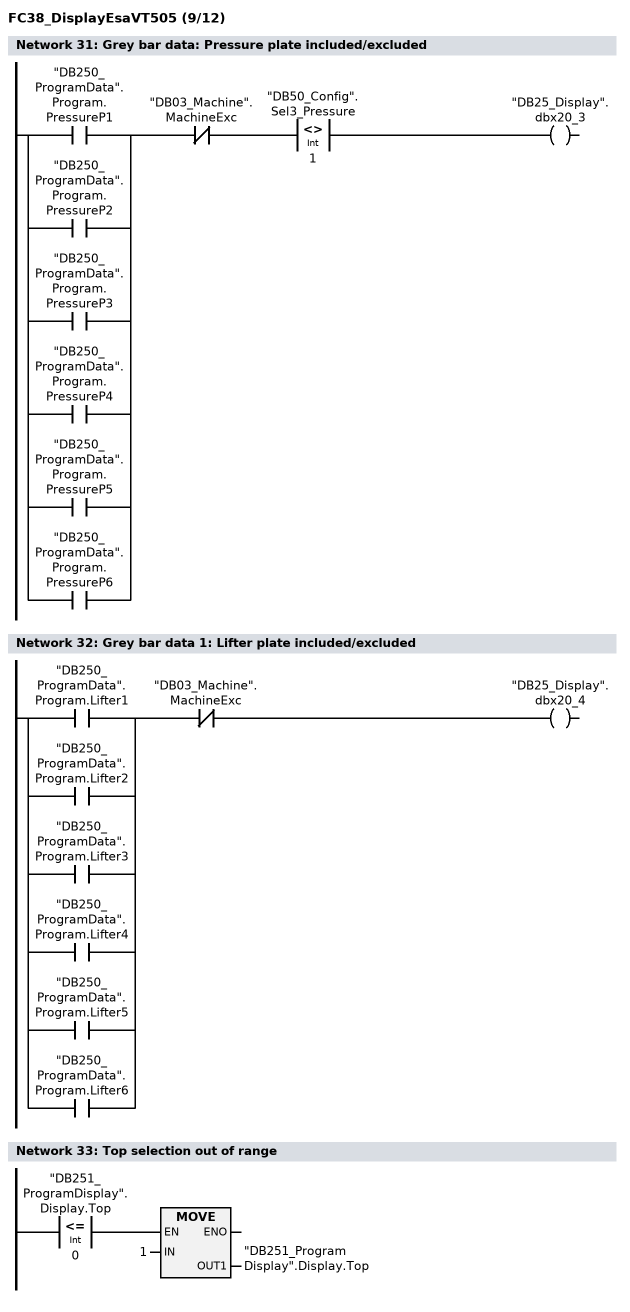
   RUNG wire#powerrail
      Contact( "DB250_ProgramData".Program.PressureP1 )
      wire#w1
      I_Contact( "DB03_Machine".MachineExc )
      { S7_Templates := "SrcType := Int" } NE_Contact(in1 := "DB50_Config".Sel3_Pressure, in2 := 1)
      Coil( "DB25_Display".dbx20_3 )
   END_RUNG
   RUNG wire#powerrail
      Contact( "DB250_ProgramData".Program.PressureP2 )
   END_RUNG wire#w1
   RUNG wire#powerrail
      Contact( "DB250_ProgramData".Program.PressureP3 )
   END_RUNG wire#w1
   RUNG wire#powerrail
      Contact( "DB250_ProgramData".Program.PressureP4 )
   END_RUNG wire#w1
   RUNG wire#powerrail
      Contact( "DB250_ProgramData".Program.PressureP5 )
   END_RUNG wire#w1
   RUNG wire#powerrail
      Contact( "DB250_ProgramData".Program.PressureP6 )
   END_RUNG wire#w1
   // the same network as SCL:
   "DB25_Display".dbx20_3 := ("DB250_ProgramData".Program.PressureP1 OR "DB250_ProgramData".Program.PressureP2 OR "DB250_ProgramData".Program.PressureP3 OR "DB250_ProgramData".Program.PressureP4 OR "DB250_ProgramData".Program.PressureP5 OR "DB250_ProgramData".Program.PressureP6) AND NOT "DB03_Machine".MachineExc AND ("DB50_Config".Sel3_Pressure <> 1);
END_REGION

REGION Network 32: Grey bar data 1: Lifter plate included/excluded
   RUNG wire#powerrail
      Contact( "DB250_ProgramData".Program.Lifter1 )
      wire#w1
      I_Contact( "DB03_Machine".MachineExc )
      Coil( "DB25_Display".dbx20_4 )
   END_RUNG
   RUNG wire#powerrail
      Contact( "DB250_ProgramData".Program.Lifter2 )
   END_RUNG wire#w1
   RUNG wire#powerrail
      Contact( "DB250_ProgramData".Program.Lifter3 )
   END_RUNG wire#w1
   RUNG wire#powerrail
      Contact( "DB250_ProgramData".Program.Lifter4 )
   END_RUNG wire#w1
   RUNG wire#powerrail
      Contact( "DB250_ProgramData".Program.Lifter5 )
   END_RUNG wire#w1
   RUNG wire#powerrail
      Contact( "DB250_ProgramData".Program.Lifter6 )
   END_RUNG wire#w1
   // the same network as SCL:
   "DB25_Display".dbx20_4 := ("DB250_ProgramData".Program.Lifter1 OR "DB250_ProgramData".Program.Lifter2 OR "DB250_ProgramData".Program.Lifter3 OR "DB250_ProgramData".Program.Lifter4 OR "DB250_ProgramData".Program.Lifter5 OR "DB250_ProgramData".Program.Lifter6) AND NOT "DB03_Machine".MachineExc;
END_REGION

REGION Network 33: Top selection out of range
   RUNG wire#powerrail
      { S7_Templates := "SrcType := Int" } LE_Contact(in1 := "DB251_ProgramDisplay".Display.Top, in2 := 0)
      { S7_GenerateENO := "TRUE" } Move(in := 1, out1 => "DB251_ProgramDisplay".Display.Top)
   END_RUNG
   // the same network as SCL:
   IF "DB251_ProgramDisplay".Display.Top <= 0 THEN "DB251_ProgramDisplay".Display.Top := 1; END_IF;
END_REGION

REGION Network 34: Top film lenght out of range
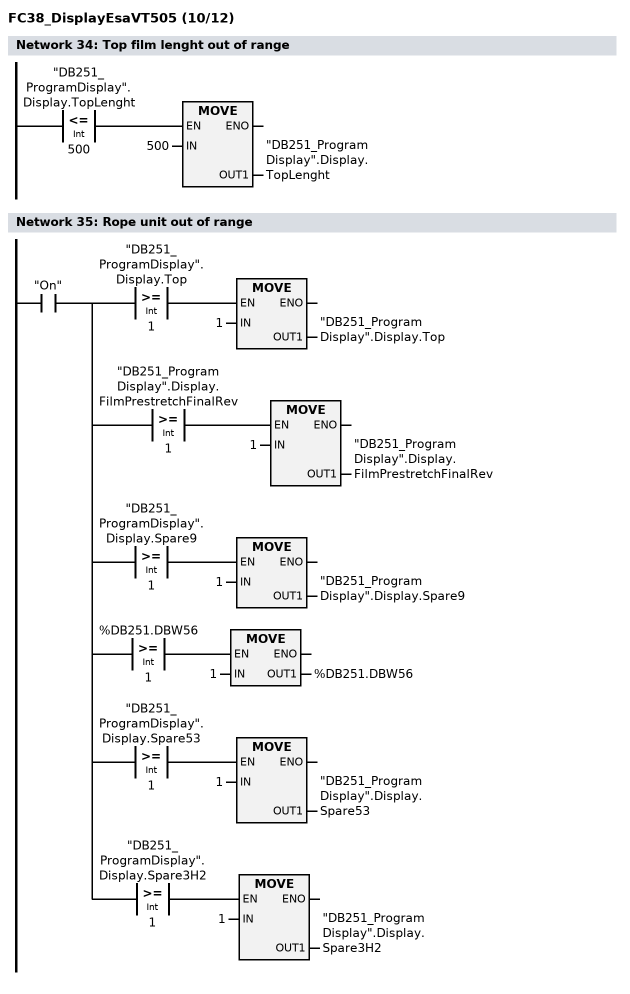
   RUNG wire#powerrail
      { S7_Templates := "SrcType := Int" } LE_Contact(in1 := "DB251_ProgramDisplay".Display.TopLenght, in2 := 500)
      { S7_GenerateENO := "TRUE" } Move(in := 500, out1 => "DB251_ProgramDisplay".Display.TopLenght)
   END_RUNG
   // the same network as SCL:
   IF "DB251_ProgramDisplay".Display.TopLenght <= 500 THEN
       "DB251_ProgramDisplay".Display.TopLenght := 500;
   END_IF;
END_REGION

REGION Network 35: Rope unit out of range
   RUNG wire#powerrail
      Contact( "On" )
      wire#w1
      { S7_Templates := "SrcType := Int" } GE_Contact(in1 := "DB251_ProgramDisplay".Display.Top, in2 := 1)
      { S7_GenerateENO := "TRUE" } Move(in := 1, out1 => "DB251_ProgramDisplay".Display.Top)
   END_RUNG
   RUNG wire#w1
      { S7_Templates := "SrcType := Int" } GE_Contact(in1 := "DB251_ProgramDisplay".Display.FilmPrestretchFinalRev, in2 := 1)
      { S7_GenerateENO := "TRUE" } Move(in := 1, out1 => "DB251_ProgramDisplay".Display.FilmPrestretchFinalRev)
   END_RUNG
   RUNG wire#w1
      { S7_Templates := "SrcType := Int" } GE_Contact(in1 := "DB251_ProgramDisplay".Display.Spare9, in2 := 1)
      { S7_GenerateENO := "TRUE" } Move(in := 1, out1 => "DB251_ProgramDisplay".Display.Spare9)
   END_RUNG
   RUNG wire#w1
      { S7_Templates := "SrcType := Int" } GE_Contact(in1 := %DB251.DBW56, in2 := 1)
      { S7_GenerateENO := "TRUE" } Move(in := 1, out1 => %DB251.DBW56)
   END_RUNG
   RUNG wire#w1
      { S7_Templates := "SrcType := Int" } GE_Contact(in1 := "DB251_ProgramDisplay".Display.Spare53, in2 := 1)
      { S7_GenerateENO := "TRUE" } Move(in := 1, out1 => "DB251_ProgramDisplay".Display.Spare53)
   END_RUNG
   RUNG wire#w1
      { S7_Templates := "SrcType := Int" } GE_Contact(in1 := "DB251_ProgramDisplay".Display.Spare3H2, in2 := 1)
      { S7_GenerateENO := "TRUE" } Move(in := 1, out1 => "DB251_ProgramDisplay".Display.Spare3H2)
   END_RUNG
   // the same network as SCL:
   IF "On" AND ("DB251_ProgramDisplay".Display.Top >= 1) THEN
       "DB251_ProgramDisplay".Display.Top := 1;
   END_IF;
   IF "On" AND ("DB251_ProgramDisplay".Display.FilmPrestretchFinalRev >= 1) THEN
       "DB251_ProgramDisplay".Display.FilmPrestretchFinalRev := 1;
   END_IF;
   IF "On" AND ("DB251_ProgramDisplay".Display.Spare9 >= 1) THEN
       "DB251_ProgramDisplay".Display.Spare9 := 1;
   END_IF;
   IF "On" AND (%DB251.DBW56 >= 1) THEN %DB251.DBW56 := 1; END_IF;
   IF "On" AND ("DB251_ProgramDisplay".Display.Spare53 >= 1) THEN
       "DB251_ProgramDisplay".Display.Spare53 := 1;
   END_IF;
   IF "On" AND ("DB251_ProgramDisplay".Display.Spare3H2 >= 1) THEN
       "DB251_ProgramDisplay".Display.Spare3H2 := 1;
   END_IF;
END_REGION

REGION Network 36: Rope unit out of range
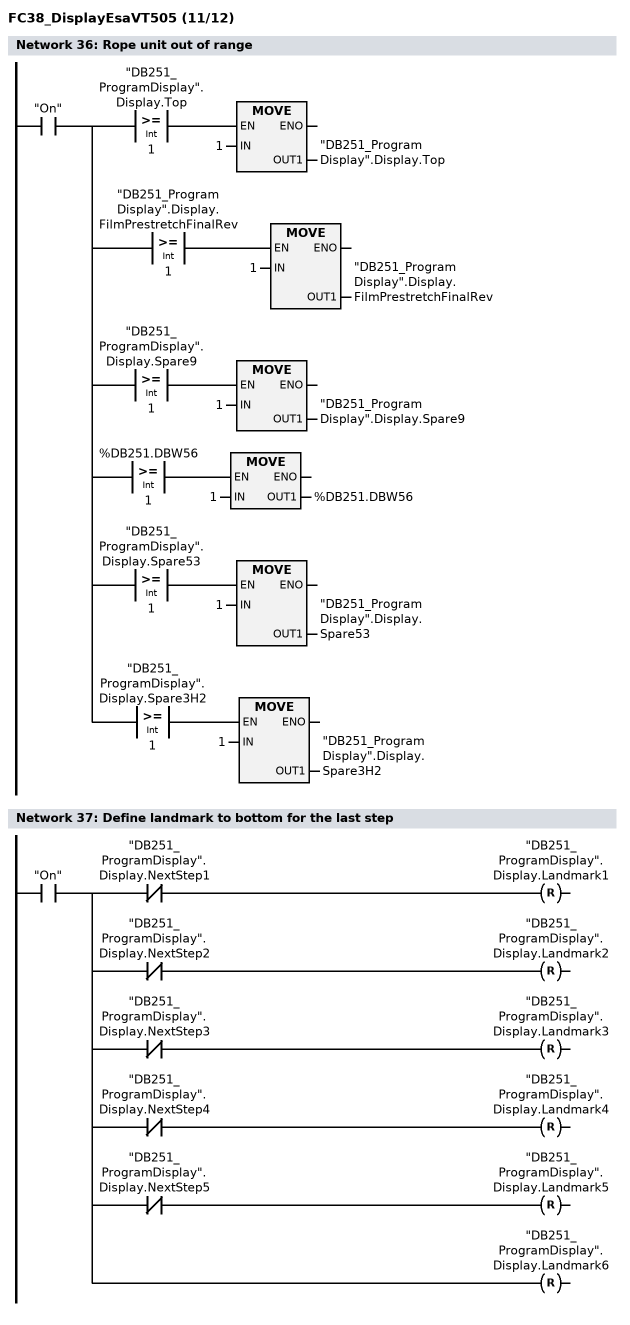
   RUNG wire#powerrail
      Contact( "On" )
      wire#w1
      { S7_Templates := "SrcType := Int" } GE_Contact(in1 := "DB251_ProgramDisplay".Display.Top, in2 := 1)
      { S7_GenerateENO := "TRUE" } Move(in := 1, out1 => "DB251_ProgramDisplay".Display.Top)
   END_RUNG
   RUNG wire#w1
      { S7_Templates := "SrcType := Int" } GE_Contact(in1 := "DB251_ProgramDisplay".Display.FilmPrestretchFinalRev, in2 := 1)
      { S7_GenerateENO := "TRUE" } Move(in := 1, out1 => "DB251_ProgramDisplay".Display.FilmPrestretchFinalRev)
   END_RUNG
   RUNG wire#w1
      { S7_Templates := "SrcType := Int" } GE_Contact(in1 := "DB251_ProgramDisplay".Display.Spare9, in2 := 1)
      { S7_GenerateENO := "TRUE" } Move(in := 1, out1 => "DB251_ProgramDisplay".Display.Spare9)
   END_RUNG
   RUNG wire#w1
      { S7_Templates := "SrcType := Int" } GE_Contact(in1 := %DB251.DBW56, in2 := 1)
      { S7_GenerateENO := "TRUE" } Move(in := 1, out1 => %DB251.DBW56)
   END_RUNG
   RUNG wire#w1
      { S7_Templates := "SrcType := Int" } GE_Contact(in1 := "DB251_ProgramDisplay".Display.Spare53, in2 := 1)
      { S7_GenerateENO := "TRUE" } Move(in := 1, out1 => "DB251_ProgramDisplay".Display.Spare53)
   END_RUNG
   RUNG wire#w1
      { S7_Templates := "SrcType := Int" } GE_Contact(in1 := "DB251_ProgramDisplay".Display.Spare3H2, in2 := 1)
      { S7_GenerateENO := "TRUE" } Move(in := 1, out1 => "DB251_ProgramDisplay".Display.Spare3H2)
   END_RUNG
   // the same network as SCL:
   IF "On" AND ("DB251_ProgramDisplay".Display.Top >= 1) THEN
       "DB251_ProgramDisplay".Display.Top := 1;
   END_IF;
   IF "On" AND ("DB251_ProgramDisplay".Display.FilmPrestretchFinalRev >= 1) THEN
       "DB251_ProgramDisplay".Display.FilmPrestretchFinalRev := 1;
   END_IF;
   IF "On" AND ("DB251_ProgramDisplay".Display.Spare9 >= 1) THEN
       "DB251_ProgramDisplay".Display.Spare9 := 1;
   END_IF;
   IF "On" AND (%DB251.DBW56 >= 1) THEN %DB251.DBW56 := 1; END_IF;
   IF "On" AND ("DB251_ProgramDisplay".Display.Spare53 >= 1) THEN
       "DB251_ProgramDisplay".Display.Spare53 := 1;
   END_IF;
   IF "On" AND ("DB251_ProgramDisplay".Display.Spare3H2 >= 1) THEN
       "DB251_ProgramDisplay".Display.Spare3H2 := 1;
   END_IF;
END_REGION

REGION Network 37: Define landmark to bottom for the last step
   RUNG wire#powerrail
      Contact( "On" )
      wire#w1
      I_Contact( "DB251_ProgramDisplay".Display.NextStep1 )
      R_Coil( "DB251_ProgramDisplay".Display.Landmark1 )
   END_RUNG
   RUNG wire#w1
      I_Contact( "DB251_ProgramDisplay".Display.NextStep2 )
      R_Coil( "DB251_ProgramDisplay".Display.Landmark2 )
   END_RUNG
   RUNG wire#w1
      I_Contact( "DB251_ProgramDisplay".Display.NextStep3 )
      R_Coil( "DB251_ProgramDisplay".Display.Landmark3 )
   END_RUNG
   RUNG wire#w1
      I_Contact( "DB251_ProgramDisplay".Display.NextStep4 )
      R_Coil( "DB251_ProgramDisplay".Display.Landmark4 )
   END_RUNG
   RUNG wire#w1
      I_Contact( "DB251_ProgramDisplay".Display.NextStep5 )
      R_Coil( "DB251_ProgramDisplay".Display.Landmark5 )
   END_RUNG
   RUNG wire#w1
      R_Coil( "DB251_ProgramDisplay".Display.Landmark6 )
   END_RUNG
   // the same network as SCL:
   IF "On" AND NOT "DB251_ProgramDisplay".Display.NextStep1 THEN
       "DB251_ProgramDisplay".Display.Landmark1 := FALSE;
   END_IF;
   IF "On" AND NOT "DB251_ProgramDisplay".Display.NextStep2 THEN
       "DB251_ProgramDisplay".Display.Landmark2 := FALSE;
   END_IF;
   IF "On" AND NOT "DB251_ProgramDisplay".Display.NextStep3 THEN
       "DB251_ProgramDisplay".Display.Landmark3 := FALSE;
   END_IF;
   IF "On" AND NOT "DB251_ProgramDisplay".Display.NextStep4 THEN
       "DB251_ProgramDisplay".Display.Landmark4 := FALSE;
   END_IF;
   IF "On" AND NOT "DB251_ProgramDisplay".Display.NextStep5 THEN
       "DB251_ProgramDisplay".Display.Landmark5 := FALSE;
   END_IF;
   IF "On" THEN "DB251_ProgramDisplay".Display.Landmark6 := FALSE; END_IF;
END_REGION

REGION Network 38
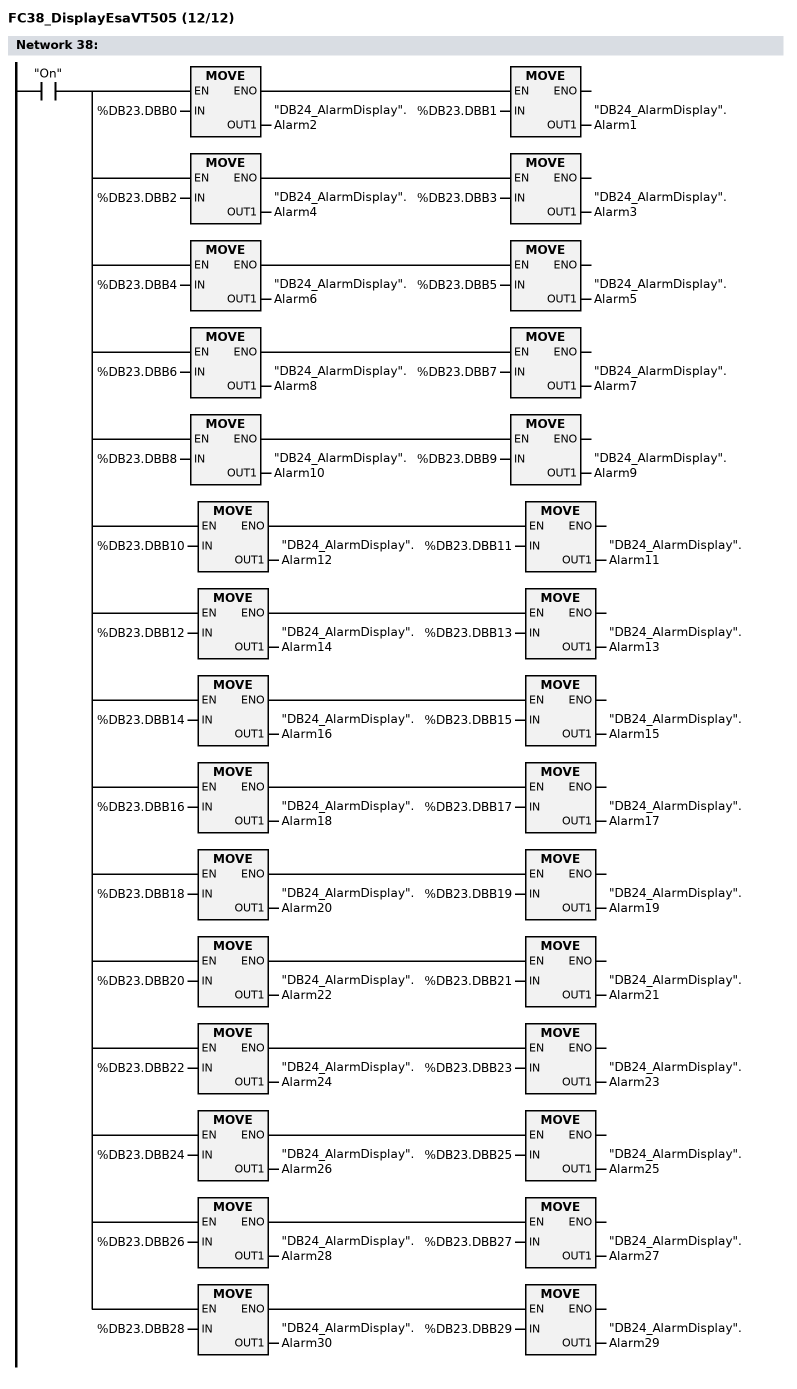
   RUNG wire#powerrail
      Contact( "On" )
      wire#w1
      { S7_GenerateENO := "TRUE" } Move(in := %DB23.DBB0, out1 => "DB24_AlarmDisplay".Alarm2)
      { S7_GenerateENO := "TRUE" } Move(in := %DB23.DBB1, out1 => "DB24_AlarmDisplay".Alarm1)
   END_RUNG
   RUNG wire#w1
      { S7_GenerateENO := "TRUE" } Move(in := %DB23.DBB2, out1 => "DB24_AlarmDisplay".Alarm4)
      { S7_GenerateENO := "TRUE" } Move(in := %DB23.DBB3, out1 => "DB24_AlarmDisplay".Alarm3)
   END_RUNG
   RUNG wire#w1
      { S7_GenerateENO := "TRUE" } Move(in := %DB23.DBB4, out1 => "DB24_AlarmDisplay".Alarm6)
      { S7_GenerateENO := "TRUE" } Move(in := %DB23.DBB5, out1 => "DB24_AlarmDisplay".Alarm5)
   END_RUNG
   RUNG wire#w1
      { S7_GenerateENO := "TRUE" } Move(in := %DB23.DBB6, out1 => "DB24_AlarmDisplay".Alarm8)
      { S7_GenerateENO := "TRUE" } Move(in := %DB23.DBB7, out1 => "DB24_AlarmDisplay".Alarm7)
   END_RUNG
   RUNG wire#w1
      { S7_GenerateENO := "TRUE" } Move(in := %DB23.DBB8, out1 => "DB24_AlarmDisplay".Alarm10)
      { S7_GenerateENO := "TRUE" } Move(in := %DB23.DBB9, out1 => "DB24_AlarmDisplay".Alarm9)
   END_RUNG
   RUNG wire#w1
      { S7_GenerateENO := "TRUE" } Move(in := %DB23.DBB10, out1 => "DB24_AlarmDisplay".Alarm12)
      { S7_GenerateENO := "TRUE" } Move(in := %DB23.DBB11, out1 => "DB24_AlarmDisplay".Alarm11)
   END_RUNG
   RUNG wire#w1
      { S7_GenerateENO := "TRUE" } Move(in := %DB23.DBB12, out1 => "DB24_AlarmDisplay".Alarm14)
      { S7_GenerateENO := "TRUE" } Move(in := %DB23.DBB13, out1 => "DB24_AlarmDisplay".Alarm13)
   END_RUNG
   RUNG wire#w1
      { S7_GenerateENO := "TRUE" } Move(in := %DB23.DBB14, out1 => "DB24_AlarmDisplay".Alarm16)
      { S7_GenerateENO := "TRUE" } Move(in := %DB23.DBB15, out1 => "DB24_AlarmDisplay".Alarm15)
   END_RUNG
   RUNG wire#w1
      { S7_GenerateENO := "TRUE" } Move(in := %DB23.DBB16, out1 => "DB24_AlarmDisplay".Alarm18)
      { S7_GenerateENO := "TRUE" } Move(in := %DB23.DBB17, out1 => "DB24_AlarmDisplay".Alarm17)
   END_RUNG
   RUNG wire#w1
      { S7_GenerateENO := "TRUE" } Move(in := %DB23.DBB18, out1 => "DB24_AlarmDisplay".Alarm20)
      { S7_GenerateENO := "TRUE" } Move(in := %DB23.DBB19, out1 => "DB24_AlarmDisplay".Alarm19)
   END_RUNG
   RUNG wire#w1
      { S7_GenerateENO := "TRUE" } Move(in := %DB23.DBB20, out1 => "DB24_AlarmDisplay".Alarm22)
      { S7_GenerateENO := "TRUE" } Move(in := %DB23.DBB21, out1 => "DB24_AlarmDisplay".Alarm21)
   END_RUNG
   RUNG wire#w1
      { S7_GenerateENO := "TRUE" } Move(in := %DB23.DBB22, out1 => "DB24_AlarmDisplay".Alarm24)
      { S7_GenerateENO := "TRUE" } Move(in := %DB23.DBB23, out1 => "DB24_AlarmDisplay".Alarm23)
   END_RUNG
   RUNG wire#w1
      { S7_GenerateENO := "TRUE" } Move(in := %DB23.DBB24, out1 => "DB24_AlarmDisplay".Alarm26)
      { S7_GenerateENO := "TRUE" } Move(in := %DB23.DBB25, out1 => "DB24_AlarmDisplay".Alarm25)
   END_RUNG
   RUNG wire#w1
      { S7_GenerateENO := "TRUE" } Move(in := %DB23.DBB26, out1 => "DB24_AlarmDisplay".Alarm28)
      { S7_GenerateENO := "TRUE" } Move(in := %DB23.DBB27, out1 => "DB24_AlarmDisplay".Alarm27)
   END_RUNG
   RUNG wire#w1
      { S7_GenerateENO := "TRUE" } Move(in := %DB23.DBB28, out1 => "DB24_AlarmDisplay".Alarm30)
      { S7_GenerateENO := "TRUE" } Move(in := %DB23.DBB29, out1 => "DB24_AlarmDisplay".Alarm29)
   END_RUNG
   // the same network as SCL:
   // ENO of a box is taken as its EN; it also drops when the box reports an error
   IF "On" THEN
       "DB24_AlarmDisplay".Alarm2 := %DB23.DBB0;
       "DB24_AlarmDisplay".Alarm1 := %DB23.DBB1;
       "DB24_AlarmDisplay".Alarm4 := %DB23.DBB2;
       "DB24_AlarmDisplay".Alarm3 := %DB23.DBB3;
       "DB24_AlarmDisplay".Alarm6 := %DB23.DBB4;
       "DB24_AlarmDisplay".Alarm5 := %DB23.DBB5;
       "DB24_AlarmDisplay".Alarm8 := %DB23.DBB6;
       "DB24_AlarmDisplay".Alarm7 := %DB23.DBB7;
       "DB24_AlarmDisplay".Alarm10 := %DB23.DBB8;
       "DB24_AlarmDisplay".Alarm9 := %DB23.DBB9;
       "DB24_AlarmDisplay".Alarm12 := %DB23.DBB10;
       "DB24_AlarmDisplay".Alarm11 := %DB23.DBB11;
       "DB24_AlarmDisplay".Alarm14 := %DB23.DBB12;
       "DB24_AlarmDisplay".Alarm13 := %DB23.DBB13;
       "DB24_AlarmDisplay".Alarm16 := %DB23.DBB14;
       "DB24_AlarmDisplay".Alarm15 := %DB23.DBB15;
       "DB24_AlarmDisplay".Alarm18 := %DB23.DBB16;
       "DB24_AlarmDisplay".Alarm17 := %DB23.DBB17;
       "DB24_AlarmDisplay".Alarm20 := %DB23.DBB18;
       "DB24_AlarmDisplay".Alarm19 := %DB23.DBB19;
       "DB24_AlarmDisplay".Alarm22 := %DB23.DBB20;
       "DB24_AlarmDisplay".Alarm21 := %DB23.DBB21;
       "DB24_AlarmDisplay".Alarm24 := %DB23.DBB22;
       "DB24_AlarmDisplay".Alarm23 := %DB23.DBB23;
       "DB24_AlarmDisplay".Alarm26 := %DB23.DBB24;
       "DB24_AlarmDisplay".Alarm25 := %DB23.DBB25;
       "DB24_AlarmDisplay".Alarm28 := %DB23.DBB26;
       "DB24_AlarmDisplay".Alarm27 := %DB23.DBB27;
       "DB24_AlarmDisplay".Alarm30 := %DB23.DBB28;
       "DB24_AlarmDisplay".Alarm29 := %DB23.DBB29;
   END_IF;
END_REGION
END_FUNCTION

FUNCTION "FC42_RopeUnit" : Void   // FC42, LAD
TITLE = RopeUnit
{ S7_Optimized_Access := 'FALSE' }
VERSION : 0.1
// stored: AutoNumber false, IsIECCheckEnabled false, SetENOAutomatically false, UDAEnableTagReadback false
   VAR_TEMP
      OpenCloseDoubleRope : Bool;
      DoubleRopeOpen : Bool;
      TempInt : Int;
      TempInt1 : Int;
   END_VAR
   VAR_TEMP   // added for the SCL form of the ladder/FBD networks
      _w1 : Bool;
   END_VAR
BEGIN

REGION Network 1: Timeout for single or lower(double) rope unit open/close
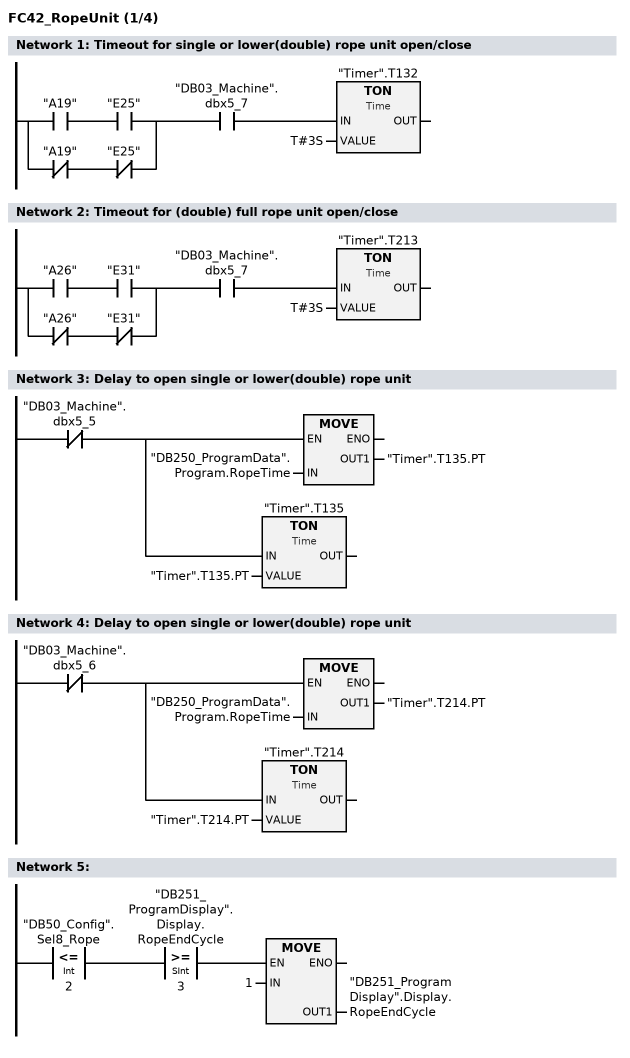
   "Timer".T132.TON(IN := (("A19" AND "E25") OR (NOT "A19" AND NOT "E25")) AND "DB03_Machine".dbx5_7, PT := T#3S);   // TON coil
END_REGION

REGION Network 2: Timeout for (double) full rope unit open/close
   "Timer".T213.TON(IN := (("A26" AND "E31") OR (NOT "A26" AND NOT "E31")) AND "DB03_Machine".dbx5_7, PT := T#3S);   // TON coil
END_REGION

REGION Network 3: Delay to open single or lower(double) rope unit
   #_w1 := NOT "DB03_Machine".dbx5_5;
   IF #_w1 THEN "Timer".T135.PT := "DB250_ProgramData".Program.RopeTime; END_IF;
   "Timer".T135.TON(IN := #_w1, PT := "Timer".T135.PT);   // TON coil
END_REGION

REGION Network 4: Delay to open single or lower(double) rope unit
   #_w1 := NOT "DB03_Machine".dbx5_6;
   IF #_w1 THEN "Timer".T214.PT := "DB250_ProgramData".Program.RopeTime; END_IF;
   "Timer".T214.TON(IN := #_w1, PT := "Timer".T214.PT);   // TON coil
END_REGION

REGION Network 5
   RUNG wire#powerrail
      { S7_Templates := "SrcType := Int" } LE_Contact(in1 := "DB50_Config".Sel8_Rope, in2 := 2)
      { S7_Templates := "SrcType := SInt" } GE_Contact(in1 := "DB251_ProgramDisplay".Display.RopeEndCycle, in2 := 3)
      { S7_GenerateENO := "TRUE" } Move(in := 1, out1 => "DB251_ProgramDisplay".Display.RopeEndCycle)
   END_RUNG
   // the same network as SCL:
   IF ("DB50_Config".Sel8_Rope <= 2) AND ("DB251_ProgramDisplay".Display.RopeEndCycle >= 3) THEN
       "DB251_ProgramDisplay".Display.RopeEndCycle := 1;
   END_IF;
END_REGION

REGION Network 6: RopeUnitOk1: Rope unit open
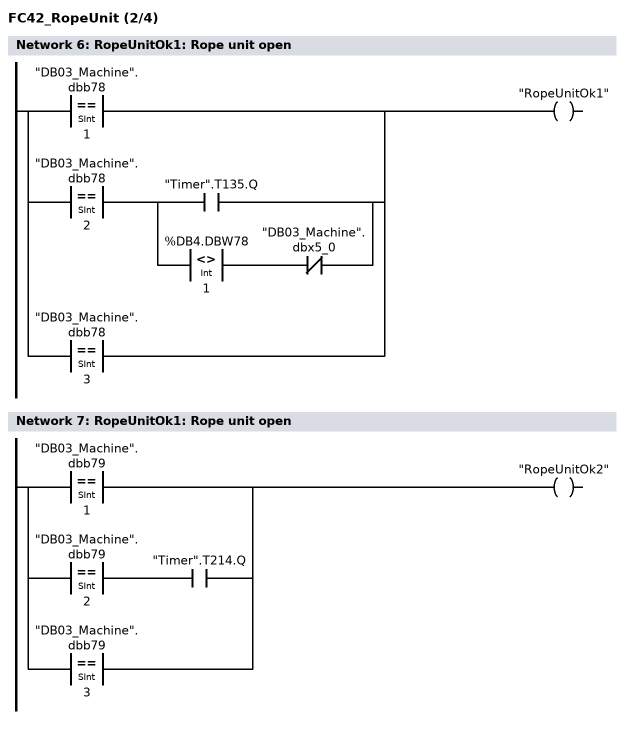
   RUNG wire#powerrail
      { S7_Templates := "SrcType := SInt" } EQ_Contact(in1 := "DB03_Machine".dbb78, in2 := 1)
      wire#w1
      Coil( "RopeUnitOk1" )
   END_RUNG
   RUNG wire#powerrail
      { S7_Templates := "SrcType := SInt" } EQ_Contact(in1 := "DB03_Machine".dbb78, in2 := 2)
      wire#w2
      Contact( "Timer".T135.Q )
   END_RUNG wire#w1
   RUNG wire#w2
      { S7_Templates := "SrcType := Int" } NE_Contact(in1 := %DB4.DBW78, in2 := 1)
      I_Contact( "DB03_Machine".dbx5_0 )
   END_RUNG wire#w1
   RUNG wire#powerrail
      { S7_Templates := "SrcType := SInt" } EQ_Contact(in1 := "DB03_Machine".dbb78, in2 := 3)
   END_RUNG wire#w1
   // the same network as SCL:
   "RopeUnitOk1" := ("DB03_Machine".dbb78 = 1) OR (("DB03_Machine".dbb78 = 2) AND ("Timer".T135.Q OR ((%DB4.DBW78 <> 1) AND NOT "DB03_Machine".dbx5_0))) OR ("DB03_Machine".dbb78 = 3);
END_REGION

REGION Network 7: RopeUnitOk1: Rope unit open
   RUNG wire#powerrail
      { S7_Templates := "SrcType := SInt" } EQ_Contact(in1 := "DB03_Machine".dbb79, in2 := 1)
      wire#w1
      Coil( "RopeUnitOk2" )
   END_RUNG
   RUNG wire#powerrail
      { S7_Templates := "SrcType := SInt" } EQ_Contact(in1 := "DB03_Machine".dbb79, in2 := 2)
      Contact( "Timer".T214.Q )
   END_RUNG wire#w1
   RUNG wire#powerrail
      { S7_Templates := "SrcType := SInt" } EQ_Contact(in1 := "DB03_Machine".dbb79, in2 := 3)
   END_RUNG wire#w1
   // the same network as SCL:
   "RopeUnitOk2" := ("DB03_Machine".dbb79 = 1) OR (("DB03_Machine".dbb79 = 2) AND "Timer".T214.Q) OR ("DB03_Machine".dbb79 = 3);
END_REGION

REGION Network 8: Closing upper(double) rope unit
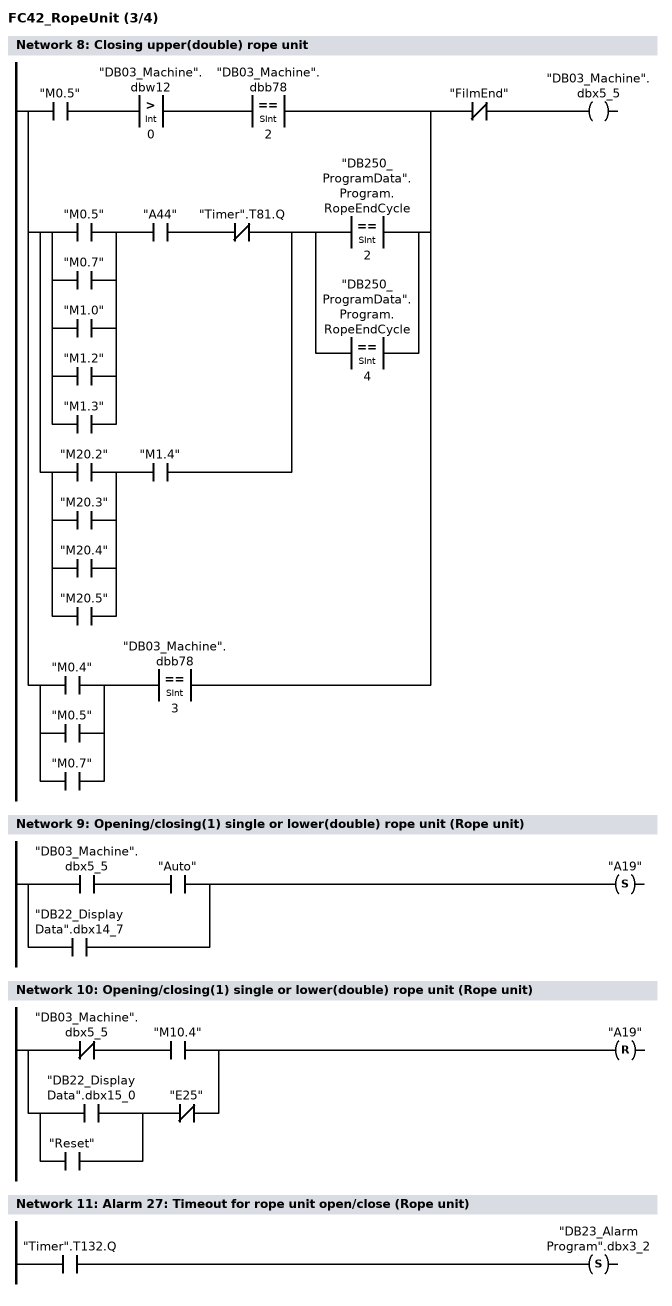
   RUNG wire#powerrail
      Contact( "M0.5" )
      { S7_Templates := "SrcType := Int" } GT_Contact(in1 := "DB03_Machine".dbw12, in2 := 0)
      { S7_Templates := "SrcType := SInt" } EQ_Contact(in1 := "DB03_Machine".dbb78, in2 := 2)
      wire#w1
      I_Contact( "FilmEnd" )
      Coil( "DB03_Machine".dbx5_5 )
   END_RUNG
   RUNG wire#powerrail
      Contact( "M0.5" )
      wire#w2
      Contact( "A44" )
      I_Contact( "Timer".T81.Q )
      wire#w3
      { S7_Templates := "SrcType := SInt" } EQ_Contact(in1 := "DB250_ProgramData".Program.RopeEndCycle, in2 := 2)
   END_RUNG wire#w1
   RUNG wire#powerrail
      Contact( "M0.7" )
   END_RUNG wire#w2
   RUNG wire#powerrail
      Contact( "M1.0" )
   END_RUNG wire#w2
   RUNG wire#powerrail
      Contact( "M1.2" )
   END_RUNG wire#w2
   RUNG wire#powerrail
      Contact( "M1.3" )
   END_RUNG wire#w2
   RUNG wire#powerrail
      Contact( "M20.2" )
      wire#w4
      Contact( "M1.4" )
   END_RUNG wire#w3
   RUNG wire#powerrail
      Contact( "M20.3" )
   END_RUNG wire#w4
   RUNG wire#powerrail
      Contact( "M20.4" )
   END_RUNG wire#w4
   RUNG wire#powerrail
      Contact( "M20.5" )
   END_RUNG wire#w4
   RUNG wire#w3
      { S7_Templates := "SrcType := SInt" } EQ_Contact(in1 := "DB250_ProgramData".Program.RopeEndCycle, in2 := 4)
   END_RUNG wire#w1
   RUNG wire#powerrail
      Contact( "M0.4" )
      wire#w5
      { S7_Templates := "SrcType := SInt" } EQ_Contact(in1 := "DB03_Machine".dbb78, in2 := 3)
   END_RUNG wire#w1
   RUNG wire#powerrail
      Contact( "M0.5" )
   END_RUNG wire#w5
   RUNG wire#powerrail
      Contact( "M0.7" )
   END_RUNG wire#w5
   // the same network as SCL:
   "DB03_Machine".dbx5_5 := (("M0.5" AND ("DB03_Machine".dbw12 > 0) AND ("DB03_Machine".dbb78 = 2)) OR (((("M0.5" OR "M0.7" OR "M1.0" OR "M1.2" OR "M1.3") AND "A44" AND NOT "Timer".T81.Q) OR (("M20.2" OR "M20.3" OR "M20.4" OR "M20.5") AND "M1.4")) AND (("DB250_ProgramData".Program.RopeEndCycle = 2) OR ("DB250_ProgramData".Program.RopeEndCycle = 4))) OR (("M0.4" OR "M0.5" OR "M0.7") AND ("DB03_Machine".dbb78 = 3))) AND NOT "FilmEnd";
END_REGION

REGION Network 9: Opening/closing(1) single or lower(double) rope unit (Rope unit)
   RUNG wire#powerrail
      Contact( "DB03_Machine".dbx5_5 )
      Contact( "Auto" )
      wire#w1
      S_Coil( "A19" )
   END_RUNG
   RUNG wire#powerrail
      Contact( "DB22_DisplayData".dbx14_7 )
   END_RUNG wire#w1
   // the same network as SCL:
   IF ("DB03_Machine".dbx5_5 AND "Auto") OR "DB22_DisplayData".dbx14_7 THEN "A19" := TRUE; END_IF;
END_REGION

REGION Network 10: Opening/closing(1) single or lower(double) rope unit (Rope unit)
   RUNG wire#powerrail
      I_Contact( "DB03_Machine".dbx5_5 )
      Contact( "M10.4" )
      wire#w1
      R_Coil( "A19" )
   END_RUNG
   RUNG wire#powerrail
      Contact( "DB22_DisplayData".dbx15_0 )
      wire#w2
      I_Contact( "E25" )
   END_RUNG wire#w1
   RUNG wire#powerrail
      Contact( "Reset" )
   END_RUNG wire#w2
   // the same network as SCL:
   IF (NOT "DB03_Machine".dbx5_5 AND "M10.4") OR (("DB22_DisplayData".dbx15_0 OR "Reset") AND NOT "E25") THEN
       "A19" := FALSE;
   END_IF;
END_REGION

REGION Network 11: Alarm 27: Timeout for rope unit open/close (Rope unit)
   RUNG wire#powerrail
      Contact( "Timer".T132.Q )
      S_Coil( "DB23_AlarmProgram".dbx3_2 )
   END_RUNG
   // the same network as SCL:
   IF "Timer".T132.Q THEN "DB23_AlarmProgram".dbx3_2 := TRUE; END_IF;
END_REGION

REGION Network 12: Closing upper(double) rope unit
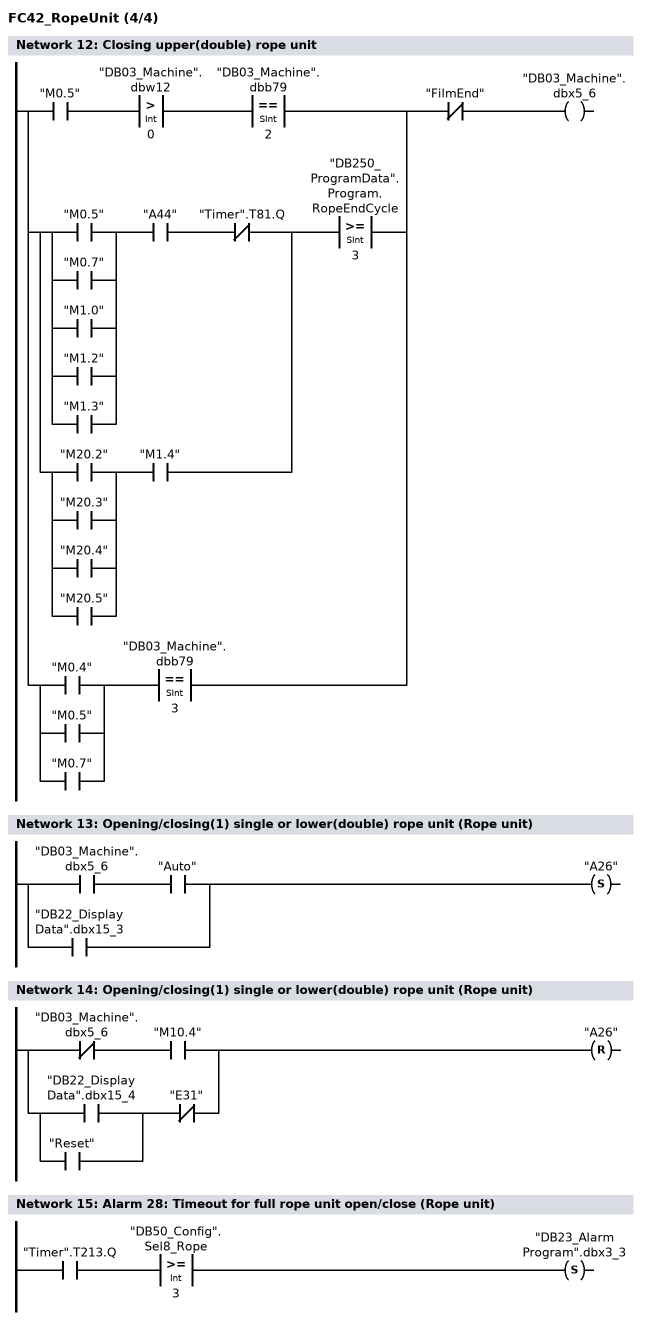
   RUNG wire#powerrail
      Contact( "M0.5" )
      { S7_Templates := "SrcType := Int" } GT_Contact(in1 := "DB03_Machine".dbw12, in2 := 0)
      { S7_Templates := "SrcType := SInt" } EQ_Contact(in1 := "DB03_Machine".dbb79, in2 := 2)
      wire#w1
      I_Contact( "FilmEnd" )
      Coil( "DB03_Machine".dbx5_6 )
   END_RUNG
   RUNG wire#powerrail
      Contact( "M0.5" )
      wire#w2
      Contact( "A44" )
      I_Contact( "Timer".T81.Q )
      wire#w3
      { S7_Templates := "SrcType := SInt" } GE_Contact(in1 := "DB250_ProgramData".Program.RopeEndCycle, in2 := 3)
   END_RUNG wire#w1
   RUNG wire#powerrail
      Contact( "M0.7" )
   END_RUNG wire#w2
   RUNG wire#powerrail
      Contact( "M1.0" )
   END_RUNG wire#w2
   RUNG wire#powerrail
      Contact( "M1.2" )
   END_RUNG wire#w2
   RUNG wire#powerrail
      Contact( "M1.3" )
   END_RUNG wire#w2
   RUNG wire#powerrail
      Contact( "M20.2" )
      wire#w4
      Contact( "M1.4" )
   END_RUNG wire#w3
   RUNG wire#powerrail
      Contact( "M20.3" )
   END_RUNG wire#w4
   RUNG wire#powerrail
      Contact( "M20.4" )
   END_RUNG wire#w4
   RUNG wire#powerrail
      Contact( "M20.5" )
   END_RUNG wire#w4
   RUNG wire#powerrail
      Contact( "M0.4" )
      wire#w5
      { S7_Templates := "SrcType := SInt" } EQ_Contact(in1 := "DB03_Machine".dbb79, in2 := 3)
   END_RUNG wire#w1
   RUNG wire#powerrail
      Contact( "M0.5" )
   END_RUNG wire#w5
   RUNG wire#powerrail
      Contact( "M0.7" )
   END_RUNG wire#w5
   // the same network as SCL:
   "DB03_Machine".dbx5_6 := (("M0.5" AND ("DB03_Machine".dbw12 > 0) AND ("DB03_Machine".dbb79 = 2)) OR (((("M0.5" OR "M0.7" OR "M1.0" OR "M1.2" OR "M1.3") AND "A44" AND NOT "Timer".T81.Q) OR (("M20.2" OR "M20.3" OR "M20.4" OR "M20.5") AND "M1.4")) AND ("DB250_ProgramData".Program.RopeEndCycle >= 3)) OR (("M0.4" OR "M0.5" OR "M0.7") AND ("DB03_Machine".dbb79 = 3))) AND NOT "FilmEnd";
END_REGION

REGION Network 13: Opening/closing(1) single or lower(double) rope unit (Rope unit)
   RUNG wire#powerrail
      Contact( "DB03_Machine".dbx5_6 )
      Contact( "Auto" )
      wire#w1
      S_Coil( "A26" )
   END_RUNG
   RUNG wire#powerrail
      Contact( "DB22_DisplayData".dbx15_3 )
   END_RUNG wire#w1
   // the same network as SCL:
   IF ("DB03_Machine".dbx5_6 AND "Auto") OR "DB22_DisplayData".dbx15_3 THEN "A26" := TRUE; END_IF;
END_REGION

REGION Network 14: Opening/closing(1) single or lower(double) rope unit (Rope unit)
   RUNG wire#powerrail
      I_Contact( "DB03_Machine".dbx5_6 )
      Contact( "M10.4" )
      wire#w1
      R_Coil( "A26" )
   END_RUNG
   RUNG wire#powerrail
      Contact( "DB22_DisplayData".dbx15_4 )
      wire#w2
      I_Contact( "E31" )
   END_RUNG wire#w1
   RUNG wire#powerrail
      Contact( "Reset" )
   END_RUNG wire#w2
   // the same network as SCL:
   IF (NOT "DB03_Machine".dbx5_6 AND "M10.4") OR (("DB22_DisplayData".dbx15_4 OR "Reset") AND NOT "E31") THEN
       "A26" := FALSE;
   END_IF;
END_REGION

REGION Network 15: Alarm 28: Timeout for full rope unit open/close (Rope unit)
   RUNG wire#powerrail
      Contact( "Timer".T213.Q )
      { S7_Templates := "SrcType := Int" } GE_Contact(in1 := "DB50_Config".Sel8_Rope, in2 := 3)
      S_Coil( "DB23_AlarmProgram".dbx3_3 )
   END_RUNG
   // the same network as SCL:
   IF "Timer".T213.Q AND ("DB50_Config".Sel8_Rope >= 3) THEN "DB23_AlarmProgram".dbx3_3 := TRUE; END_IF;
END_REGION
END_FUNCTION

FUNCTION "FC45_PrestretchPGSM_PGSA" : Void   // FC45, LAD
TITLE = Prestretch PGSM and PGSA management (HS30, Helix One)
{ S7_Optimized_Access := 'FALSE' }
AUTHOR : Robopac
VERSION : 0.0
// stored: AutoNumber false, IsIECCheckEnabled false, SetENOAutomatically false, UDAEnableTagReadback false
   VAR_TEMP
      TempInt : Int;
      TempDint : DInt;
      TempDint_2 : DInt;
      TiroStepTemp : Int;
      TiroFineTemp : Int;
   END_VAR
   VAR_TEMP   // added for the SCL form of the ladder/FBD networks
      _w1 : Bool;
      _w2 : Bool;
      _w3 : Bool;
      _w4 : Bool;
      _w5 : Bool;
      _w6 : Bool;
      _w7 : Bool;
   END_VAR
BEGIN

REGION Network 1: Film broken delay for spool carriage
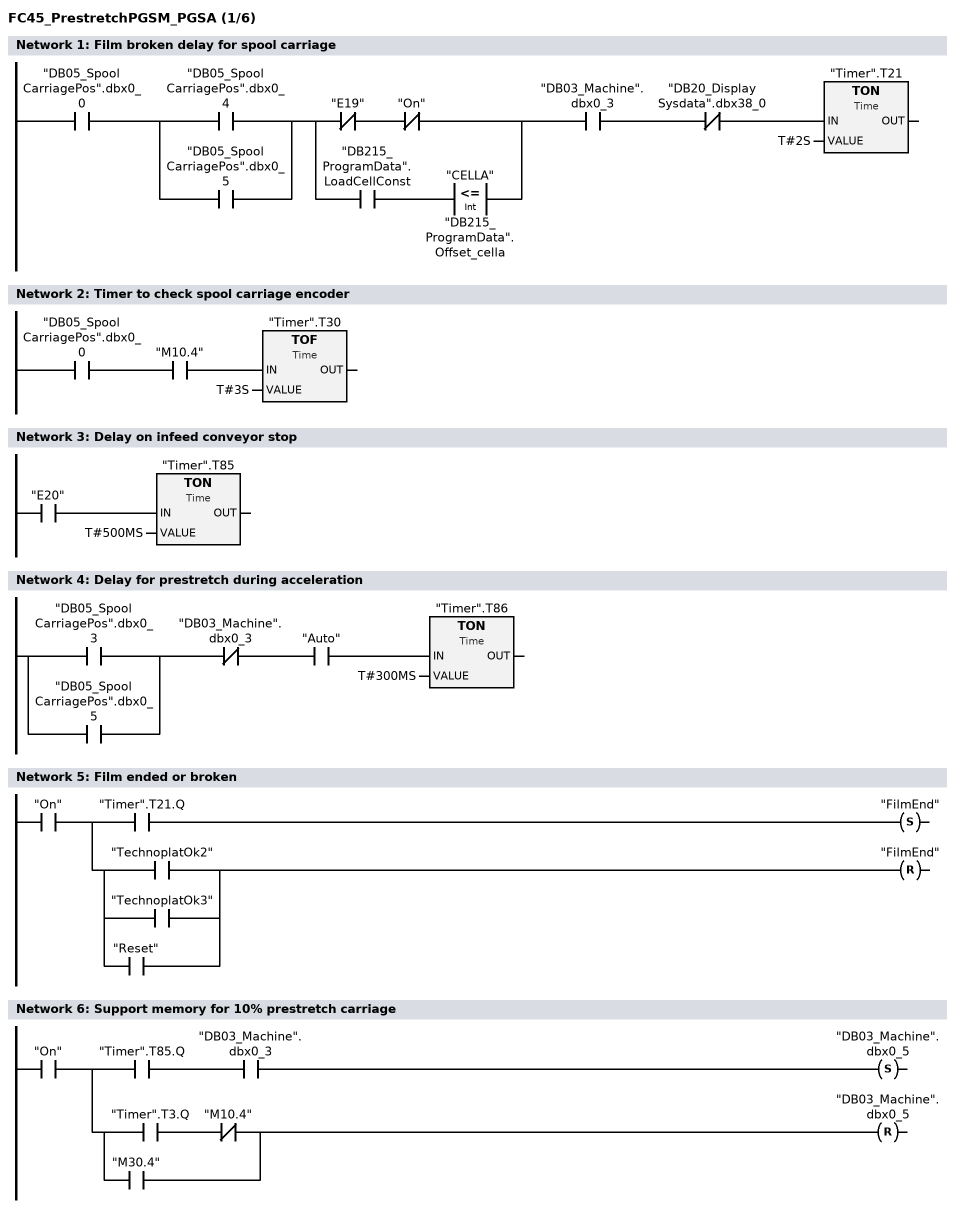
   "Timer".T21.TON(IN := "DB05_SpoolCarriagePos".dbx0_0 AND ("DB05_SpoolCarriagePos".dbx0_4 OR "DB05_SpoolCarriagePos".dbx0_5) AND ((NOT "E19" AND NOT "On") OR ("DB215_ProgramData".LoadCellConst AND ("CELLA" <= "DB215_ProgramData".Offset_cella))) AND "DB03_Machine".dbx0_3 AND NOT "DB20_DisplaySysdata".dbx38_0, PT := T#2S);   // TON coil
END_REGION

REGION Network 2: Timer to check spool carriage encoder
   "Timer".T30.TOF(IN := "DB05_SpoolCarriagePos".dbx0_0 AND "M10.4", PT := T#3S);   // TOF coil
END_REGION

REGION Network 3: Delay on infeed conveyor stop
   "Timer".T85.TON(IN := "E20", PT := T#500MS);   // TON coil
END_REGION

REGION Network 4: Delay for prestretch during acceleration
   "Timer".T86.TON(IN := ("DB05_SpoolCarriagePos".dbx0_3 OR "DB05_SpoolCarriagePos".dbx0_5) AND NOT "DB03_Machine".dbx0_3 AND "Auto", PT := T#300MS);   // TON coil
END_REGION

REGION Network 5: Film ended or broken
   RUNG wire#powerrail
      Contact( "On" )
      wire#w1
      Contact( "Timer".T21.Q )
      S_Coil( "FilmEnd" )
   END_RUNG
   RUNG wire#w1
      Contact( "TechnoplatOk2" )
      wire#w2
      R_Coil( "FilmEnd" )
   END_RUNG
   RUNG wire#w1
      Contact( "TechnoplatOk3" )
   END_RUNG wire#w2
   RUNG wire#w1
      Contact( "Reset" )
   END_RUNG wire#w2
   // the same network as SCL:
   IF "On" AND "Timer".T21.Q THEN "FilmEnd" := TRUE; END_IF;
   IF "On" AND ("TechnoplatOk2" OR "TechnoplatOk3" OR "Reset") THEN "FilmEnd" := FALSE; END_IF;
END_REGION

REGION Network 6: Support memory for 10% prestretch carriage
   RUNG wire#powerrail
      Contact( "On" )
      wire#w1
      Contact( "Timer".T85.Q )
      Contact( "DB03_Machine".dbx0_3 )
      S_Coil( "DB03_Machine".dbx0_5 )
   END_RUNG
   RUNG wire#w1
      Contact( "Timer".T3.Q )
      I_Contact( "M10.4" )
      wire#w2
      R_Coil( "DB03_Machine".dbx0_5 )
   END_RUNG
   RUNG wire#w1
      Contact( "M30.4" )
   END_RUNG wire#w2
   // the same network as SCL:
   IF "On" AND "Timer".T85.Q AND "DB03_Machine".dbx0_3 THEN "DB03_Machine".dbx0_5 := TRUE; END_IF;
   IF "On" AND (("Timer".T3.Q AND NOT "M10.4") OR "M30.4") THEN "DB03_Machine".dbx0_5 := FALSE; END_IF;
END_REGION

REGION Network 7: Support memory for prestretch PGSM or PGSA
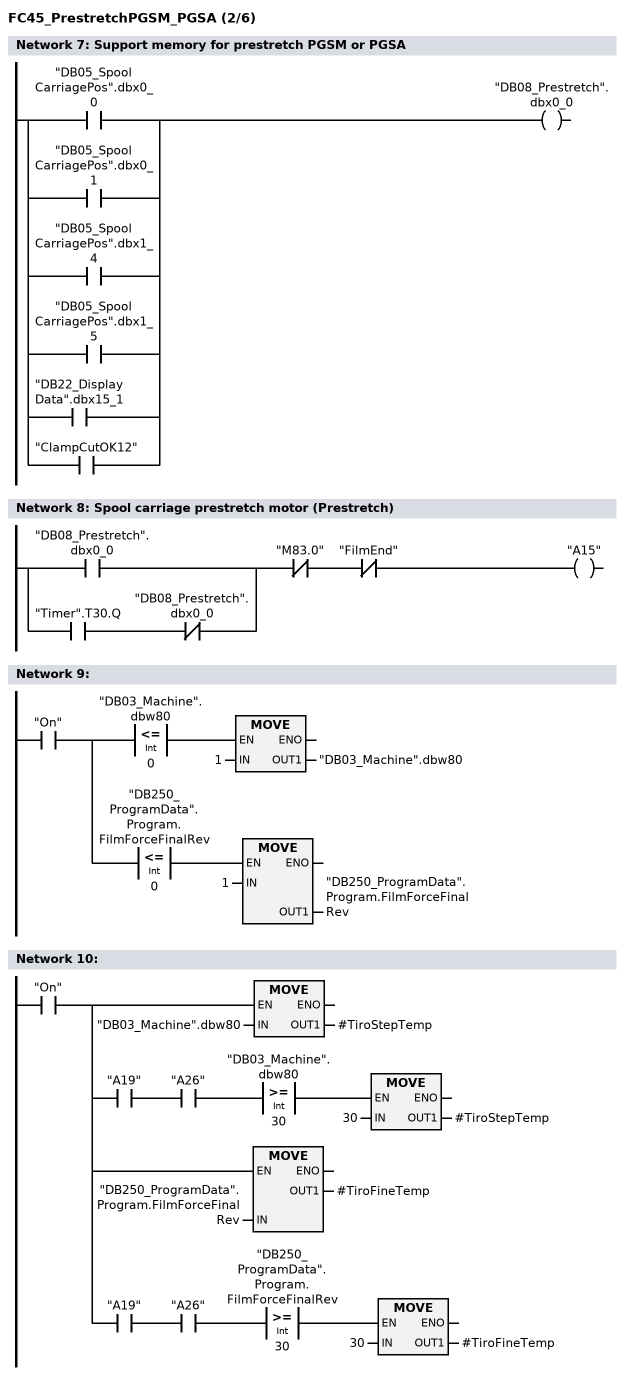
   RUNG wire#powerrail
      Contact( "DB05_SpoolCarriagePos".dbx0_0 )
      wire#w1
      Coil( "DB08_Prestretch".dbx0_0 )
   END_RUNG
   RUNG wire#powerrail
      Contact( "DB05_SpoolCarriagePos".dbx0_1 )
   END_RUNG wire#w1
   RUNG wire#powerrail
      Contact( "DB05_SpoolCarriagePos".dbx1_4 )
   END_RUNG wire#w1
   RUNG wire#powerrail
      Contact( "DB05_SpoolCarriagePos".dbx1_5 )
   END_RUNG wire#w1
   RUNG wire#powerrail
      Contact( "DB22_DisplayData".dbx15_1 )
   END_RUNG wire#w1
   RUNG wire#powerrail
      Contact( "ClampCutOK12" )
   END_RUNG wire#w1
   // the same network as SCL:
   "DB08_Prestretch".dbx0_0 := "DB05_SpoolCarriagePos".dbx0_0 OR "DB05_SpoolCarriagePos".dbx0_1 OR "DB05_SpoolCarriagePos".dbx1_4 OR "DB05_SpoolCarriagePos".dbx1_5 OR "DB22_DisplayData".dbx15_1 OR "ClampCutOK12";
END_REGION

REGION Network 8: Spool carriage prestretch motor (Prestretch)
   RUNG wire#powerrail
      Contact( "DB08_Prestretch".dbx0_0 )
      wire#w1
      I_Contact( "M83.0" )
      I_Contact( "FilmEnd" )
      Coil( "A15" )
   END_RUNG
   RUNG wire#powerrail
      Contact( "Timer".T30.Q )
      I_Contact( "DB08_Prestretch".dbx0_0 )
   END_RUNG wire#w1
   // the same network as SCL:
   "A15" := ("DB08_Prestretch".dbx0_0 OR ("Timer".T30.Q AND NOT "DB08_Prestretch".dbx0_0)) AND NOT "M83.0" AND NOT "FilmEnd";
END_REGION

REGION Network 9
   RUNG wire#powerrail
      Contact( "On" )
      wire#w1
      { S7_Templates := "SrcType := Int" } LE_Contact(in1 := "DB03_Machine".dbw80, in2 := 0)
      { S7_GenerateENO := "TRUE" } Move(in := 1, out1 => "DB03_Machine".dbw80)
   END_RUNG
   RUNG wire#w1
      { S7_Templates := "SrcType := Int" } LE_Contact(in1 := "DB250_ProgramData".Program.FilmForceFinalRev, in2 := 0)
      { S7_GenerateENO := "TRUE" } Move(in := 1, out1 => "DB250_ProgramData".Program.FilmForceFinalRev)
   END_RUNG
   // the same network as SCL:
   IF "On" AND ("DB03_Machine".dbw80 <= 0) THEN "DB03_Machine".dbw80 := 1; END_IF;
   IF "On" AND ("DB250_ProgramData".Program.FilmForceFinalRev <= 0) THEN
       "DB250_ProgramData".Program.FilmForceFinalRev := 1;
   END_IF;
END_REGION

REGION Network 10
   RUNG wire#powerrail
      Contact( "On" )
      wire#w1
      { S7_GenerateENO := "TRUE" } Move(in := "DB03_Machine".dbw80, out1 => #TiroStepTemp)
   END_RUNG
   RUNG wire#w1
      Contact( "A19" )
      Contact( "A26" )
      { S7_Templates := "SrcType := Int" } GE_Contact(in1 := "DB03_Machine".dbw80, in2 := 30)
      { S7_GenerateENO := "TRUE" } Move(in := 30, out1 => #TiroStepTemp)
   END_RUNG
   RUNG wire#w1
      { S7_GenerateENO := "TRUE" } Move(in := "DB250_ProgramData".Program.FilmForceFinalRev, out1 => #TiroFineTemp)
   END_RUNG
   RUNG wire#w1
      Contact( "A19" )
      Contact( "A26" )
      { S7_Templates := "SrcType := Int" } GE_Contact(in1 := "DB250_ProgramData".Program.FilmForceFinalRev, in2 := 30)
      { S7_GenerateENO := "TRUE" } Move(in := 30, out1 => #TiroFineTemp)
   END_RUNG
   // the same network as SCL:
   IF "On" THEN #TiroStepTemp := "DB03_Machine".dbw80; END_IF;
   IF "On" AND "A19" AND "A26" AND ("DB03_Machine".dbw80 >= 30) THEN #TiroStepTemp := 30; END_IF;
   IF "On" THEN #TiroFineTemp := "DB250_ProgramData".Program.FilmForceFinalRev; END_IF;
   IF "On" AND "A19" AND "A26" AND ("DB250_ProgramData".Program.FilmForceFinalRev >= 30) THEN
       #TiroFineTemp := 30;
   END_IF;
END_REGION

REGION Network 11
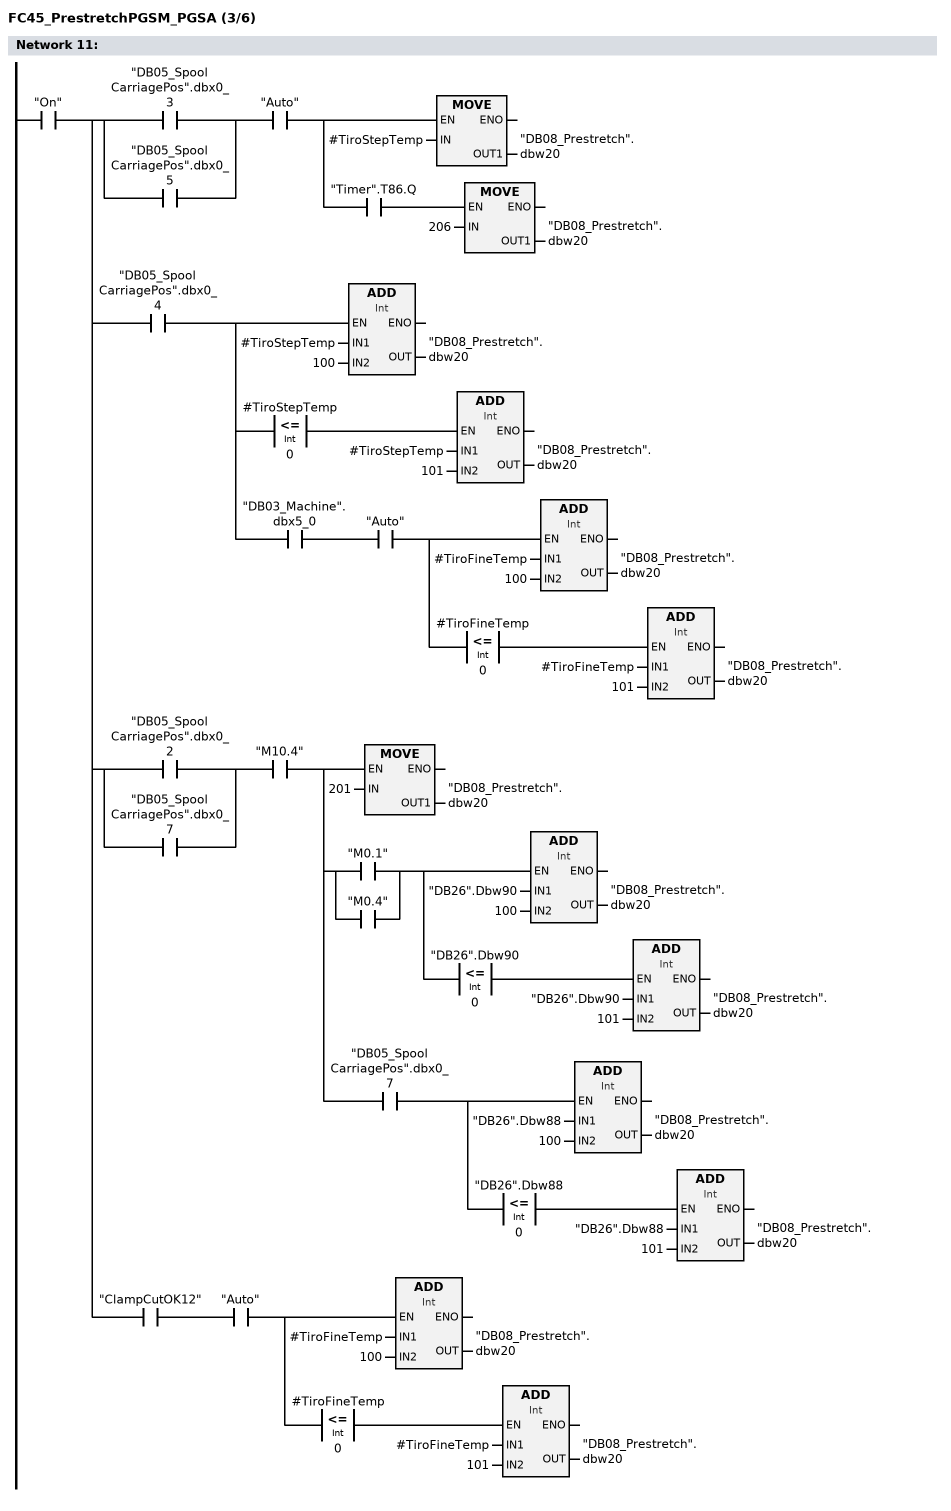
   RUNG wire#powerrail
      Contact( "On" )
      wire#w1
      Contact( "DB05_SpoolCarriagePos".dbx0_3 )
      wire#w2
      Contact( "Auto" )
      wire#w3
      { S7_GenerateENO := "TRUE" } Move(in := #TiroStepTemp, out1 => "DB08_Prestretch".dbw20)
   END_RUNG
   RUNG wire#w1
      Contact( "DB05_SpoolCarriagePos".dbx0_5 )
   END_RUNG wire#w2
   RUNG wire#w3
      Contact( "Timer".T86.Q )
      { S7_GenerateENO := "TRUE" } Move(in := 206, out1 => "DB08_Prestretch".dbw20)
   END_RUNG
   RUNG wire#w1
      Contact( "DB05_SpoolCarriagePos".dbx0_4 )
      wire#w4
      { S7_Templates := "SrcType := Int"; S7_GenerateENO := "TRUE" } Add(in1 := #TiroStepTemp, in2 := 100, out => "DB08_Prestretch".dbw20)
   END_RUNG
   RUNG wire#w4
      { S7_Templates := "SrcType := Int" } LE_Contact(in1 := #TiroStepTemp, in2 := 0)
      { S7_Templates := "SrcType := Int"; S7_GenerateENO := "TRUE" } Add(in1 := #TiroStepTemp, in2 := 101, out => "DB08_Prestretch".dbw20)
   END_RUNG
   RUNG wire#w4
      Contact( "DB03_Machine".dbx5_0 )
      Contact( "Auto" )
      wire#w5
      { S7_Templates := "SrcType := Int"; S7_GenerateENO := "TRUE" } Add(in1 := #TiroFineTemp, in2 := 100, out => "DB08_Prestretch".dbw20)
   END_RUNG
   RUNG wire#w5
      { S7_Templates := "SrcType := Int" } LE_Contact(in1 := #TiroFineTemp, in2 := 0)
      { S7_Templates := "SrcType := Int"; S7_GenerateENO := "TRUE" } Add(in1 := #TiroFineTemp, in2 := 101, out => "DB08_Prestretch".dbw20)
   END_RUNG
   RUNG wire#w1
      Contact( "DB05_SpoolCarriagePos".dbx0_2 )
      wire#w6
      Contact( "M10.4" )
      wire#w7
      { S7_GenerateENO := "TRUE" } Move(in := 201, out1 => "DB08_Prestretch".dbw20)
   END_RUNG
   RUNG wire#w1
      Contact( "DB05_SpoolCarriagePos".dbx0_7 )
   END_RUNG wire#w6
   RUNG wire#w7
      Contact( "M0.1" )
      wire#w8
      { S7_Templates := "SrcType := Int"; S7_GenerateENO := "TRUE" } Add(in1 := "DB26".Dbw90, in2 := 100, out => "DB08_Prestretch".dbw20)
   END_RUNG
   RUNG wire#w7
      Contact( "M0.4" )
   END_RUNG wire#w8
   RUNG wire#w8
      { S7_Templates := "SrcType := Int" } LE_Contact(in1 := "DB26".Dbw90, in2 := 0)
      { S7_Templates := "SrcType := Int"; S7_GenerateENO := "TRUE" } Add(in1 := "DB26".Dbw90, in2 := 101, out => "DB08_Prestretch".dbw20)
   END_RUNG
   RUNG wire#w7
      Contact( "DB05_SpoolCarriagePos".dbx0_7 )
      wire#w9
      { S7_Templates := "SrcType := Int"; S7_GenerateENO := "TRUE" } Add(in1 := "DB26".Dbw88, in2 := 100, out => "DB08_Prestretch".dbw20)
   END_RUNG
   RUNG wire#w9
      { S7_Templates := "SrcType := Int" } LE_Contact(in1 := "DB26".Dbw88, in2 := 0)
      { S7_Templates := "SrcType := Int"; S7_GenerateENO := "TRUE" } Add(in1 := "DB26".Dbw88, in2 := 101, out => "DB08_Prestretch".dbw20)
   END_RUNG
   RUNG wire#w1
      Contact( "ClampCutOK12" )
      Contact( "Auto" )
      wire#w10
      { S7_Templates := "SrcType := Int"; S7_GenerateENO := "TRUE" } Add(in1 := #TiroFineTemp, in2 := 100, out => "DB08_Prestretch".dbw20)
   END_RUNG
   RUNG wire#w10
      { S7_Templates := "SrcType := Int" } LE_Contact(in1 := #TiroFineTemp, in2 := 0)
      { S7_Templates := "SrcType := Int"; S7_GenerateENO := "TRUE" } Add(in1 := #TiroFineTemp, in2 := 101, out => "DB08_Prestretch".dbw20)
   END_RUNG
   // the same network as SCL:
   #_w1 := "On" AND ("DB05_SpoolCarriagePos".dbx0_3 OR "DB05_SpoolCarriagePos".dbx0_5) AND "Auto";
   IF #_w1 THEN "DB08_Prestretch".dbw20 := #TiroStepTemp; END_IF;
   IF #_w1 AND "Timer".T86.Q THEN "DB08_Prestretch".dbw20 := 206; END_IF;
   #_w2 := "On" AND "DB05_SpoolCarriagePos".dbx0_4;
   IF #_w2 THEN "DB08_Prestretch".dbw20 := #TiroStepTemp + 100; END_IF;
   IF #_w2 AND (#TiroStepTemp <= 0) THEN "DB08_Prestretch".dbw20 := #TiroStepTemp + 101; END_IF;
   #_w3 := #_w2 AND "DB03_Machine".dbx5_0 AND "Auto";
   IF #_w3 THEN "DB08_Prestretch".dbw20 := #TiroFineTemp + 100; END_IF;
   IF #_w3 AND (#TiroFineTemp <= 0) THEN "DB08_Prestretch".dbw20 := #TiroFineTemp + 101; END_IF;
   #_w4 := "On" AND ("DB05_SpoolCarriagePos".dbx0_2 OR "DB05_SpoolCarriagePos".dbx0_7) AND "M10.4";
   IF #_w4 THEN "DB08_Prestretch".dbw20 := 201; END_IF;
   #_w5 := #_w4 AND ("M0.1" OR "M0.4");
   IF #_w5 THEN "DB08_Prestretch".dbw20 := "DB26".Dbw90 + 100; END_IF;
   IF #_w5 AND ("DB26".Dbw90 <= 0) THEN "DB08_Prestretch".dbw20 := "DB26".Dbw90 + 101; END_IF;
   #_w6 := #_w4 AND "DB05_SpoolCarriagePos".dbx0_7;
   IF #_w6 THEN "DB08_Prestretch".dbw20 := "DB26".Dbw88 + 100; END_IF;
   IF #_w6 AND ("DB26".Dbw88 <= 0) THEN "DB08_Prestretch".dbw20 := "DB26".Dbw88 + 101; END_IF;
   #_w7 := "On" AND "ClampCutOK12" AND "Auto";
   IF #_w7 THEN "DB08_Prestretch".dbw20 := #TiroFineTemp + 100; END_IF;
   IF #_w7 AND (#TiroFineTemp <= 0) THEN "DB08_Prestretch".dbw20 := #TiroFineTemp + 101; END_IF;
END_REGION

REGION Network 12
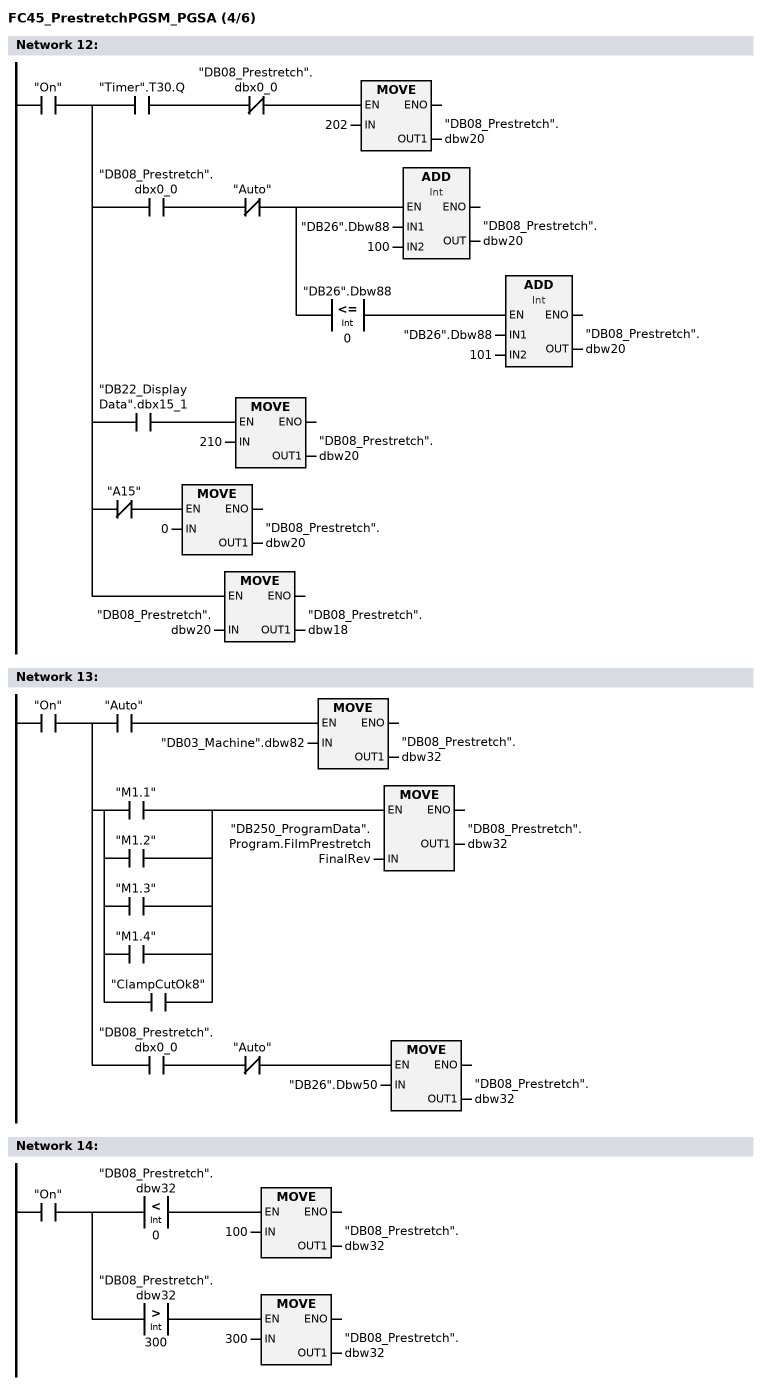
   RUNG wire#powerrail
      Contact( "On" )
      wire#w1
      Contact( "Timer".T30.Q )
      I_Contact( "DB08_Prestretch".dbx0_0 )
      { S7_GenerateENO := "TRUE" } Move(in := 202, out1 => "DB08_Prestretch".dbw20)
   END_RUNG
   RUNG wire#w1
      Contact( "DB08_Prestretch".dbx0_0 )
      I_Contact( "Auto" )
      wire#w2
      { S7_Templates := "SrcType := Int"; S7_GenerateENO := "TRUE" } Add(in1 := "DB26".Dbw88, in2 := 100, out => "DB08_Prestretch".dbw20)
   END_RUNG
   RUNG wire#w2
      { S7_Templates := "SrcType := Int" } LE_Contact(in1 := "DB26".Dbw88, in2 := 0)
      { S7_Templates := "SrcType := Int"; S7_GenerateENO := "TRUE" } Add(in1 := "DB26".Dbw88, in2 := 101, out => "DB08_Prestretch".dbw20)
   END_RUNG
   RUNG wire#w1
      Contact( "DB22_DisplayData".dbx15_1 )
      { S7_GenerateENO := "TRUE" } Move(in := 210, out1 => "DB08_Prestretch".dbw20)
   END_RUNG
   RUNG wire#w1
      I_Contact( "A15" )
      { S7_GenerateENO := "TRUE" } Move(in := 0, out1 => "DB08_Prestretch".dbw20)
   END_RUNG
   RUNG wire#w1
      { S7_GenerateENO := "TRUE" } Move(in := "DB08_Prestretch".dbw20, out1 => "DB08_Prestretch".dbw18)
   END_RUNG
   // the same network as SCL:
   IF "On" AND "Timer".T30.Q AND NOT "DB08_Prestretch".dbx0_0 THEN "DB08_Prestretch".dbw20 := 202; END_IF;
   #_w1 := "On" AND "DB08_Prestretch".dbx0_0 AND NOT "Auto";
   IF #_w1 THEN "DB08_Prestretch".dbw20 := "DB26".Dbw88 + 100; END_IF;
   IF #_w1 AND ("DB26".Dbw88 <= 0) THEN "DB08_Prestretch".dbw20 := "DB26".Dbw88 + 101; END_IF;
   IF "On" AND "DB22_DisplayData".dbx15_1 THEN "DB08_Prestretch".dbw20 := 210; END_IF;
   IF "On" AND NOT "A15" THEN "DB08_Prestretch".dbw20 := 0; END_IF;
   IF "On" THEN "DB08_Prestretch".dbw18 := "DB08_Prestretch".dbw20; END_IF;
END_REGION

REGION Network 13
   RUNG wire#powerrail
      Contact( "On" )
      wire#w1
      Contact( "Auto" )
      { S7_GenerateENO := "TRUE" } Move(in := "DB03_Machine".dbw82, out1 => "DB08_Prestretch".dbw32)
   END_RUNG
   RUNG wire#w1
      Contact( "M1.1" )
      wire#w2
      { S7_GenerateENO := "TRUE" } Move(in := "DB250_ProgramData".Program.FilmPrestretchFinalRev, out1 => "DB08_Prestretch".dbw32)
   END_RUNG
   RUNG wire#w1
      Contact( "M1.2" )
   END_RUNG wire#w2
   RUNG wire#w1
      Contact( "M1.3" )
   END_RUNG wire#w2
   RUNG wire#w1
      Contact( "M1.4" )
   END_RUNG wire#w2
   RUNG wire#w1
      Contact( "ClampCutOk8" )
   END_RUNG wire#w2
   RUNG wire#w1
      Contact( "DB08_Prestretch".dbx0_0 )
      I_Contact( "Auto" )
      { S7_GenerateENO := "TRUE" } Move(in := "DB26".Dbw50, out1 => "DB08_Prestretch".dbw32)
   END_RUNG
   // the same network as SCL:
   IF "On" AND "Auto" THEN "DB08_Prestretch".dbw32 := "DB03_Machine".dbw82; END_IF;
   IF "On" AND ("M1.1" OR "M1.2" OR "M1.3" OR "M1.4" OR "ClampCutOk8") THEN
       "DB08_Prestretch".dbw32 := "DB250_ProgramData".Program.FilmPrestretchFinalRev;
   END_IF;
   IF "On" AND "DB08_Prestretch".dbx0_0 AND NOT "Auto" THEN "DB08_Prestretch".dbw32 := "DB26".Dbw50; END_IF;
END_REGION

REGION Network 14
   RUNG wire#powerrail
      Contact( "On" )
      wire#w1
      { S7_Templates := "SrcType := Int" } LT_Contact(in1 := "DB08_Prestretch".dbw32, in2 := 0)
      { S7_GenerateENO := "TRUE" } Move(in := 100, out1 => "DB08_Prestretch".dbw32)
   END_RUNG
   RUNG wire#w1
      { S7_Templates := "SrcType := Int" } GT_Contact(in1 := "DB08_Prestretch".dbw32, in2 := 300)
      { S7_GenerateENO := "TRUE" } Move(in := 300, out1 => "DB08_Prestretch".dbw32)
   END_RUNG
   // the same network as SCL:
   IF "On" AND ("DB08_Prestretch".dbw32 < 0) THEN "DB08_Prestretch".dbw32 := 100; END_IF;
   IF "On" AND ("DB08_Prestretch".dbw32 > 300) THEN "DB08_Prestretch".dbw32 := 300; END_IF;
END_REGION

REGION Network 15
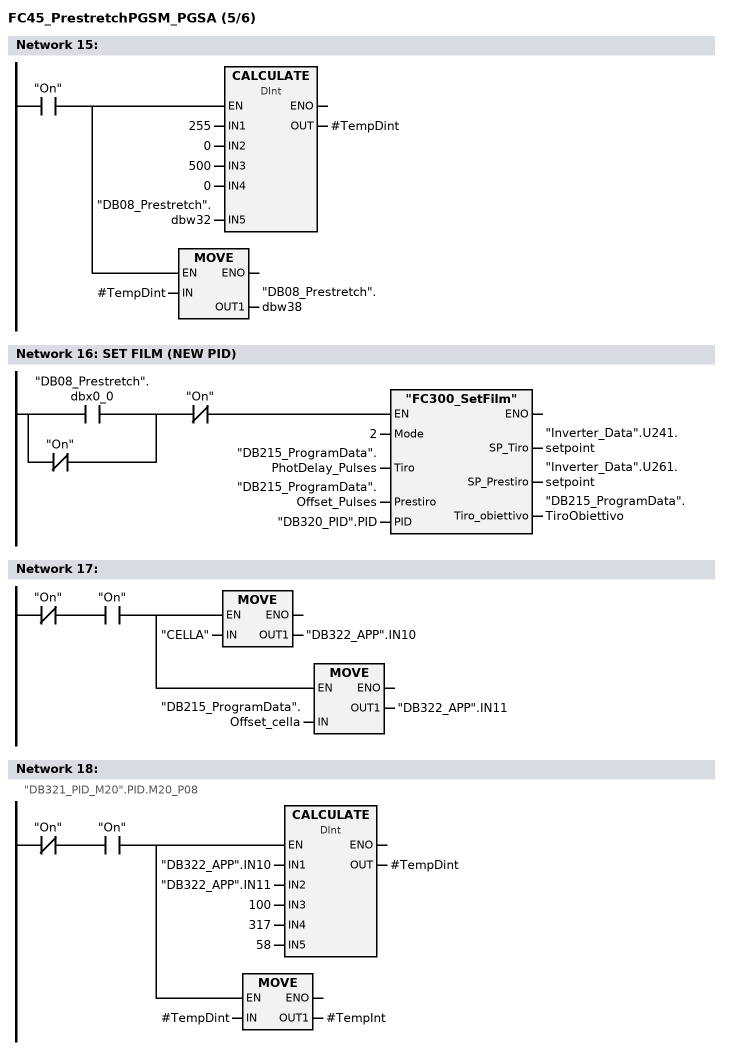
   RUNG wire#powerrail
      Contact( "On" )
      wire#w1
      { S7_Templates := "SrcType := DInt"; S7_GenerateENO := "TRUE"; S7_Expression := "((IN5-IN4)*(IN1-IN2)/(IN3-IN4))+IN2" } Calculate(in1 := 255, in2 := 0, in3 := 500, in4 := 0, in5 := "DB08_Prestretch".dbw32, out => #TempDint)
   END_RUNG
   RUNG wire#w1
      { S7_GenerateENO := "TRUE" } Move(in := #TempDint, out1 => "DB08_Prestretch".dbw38)
   END_RUNG
   // the same network as SCL:
   IF "On" THEN
       #TempDint := (("DB08_Prestretch".dbw32-0)*(255-0)/(500-0))+0;
       "DB08_Prestretch".dbw38 := #TempDint;
   END_IF;
END_REGION

REGION Network 16: SET FILM (NEW PID)
   RUNG wire#powerrail
      Contact( "DB08_Prestretch".dbx0_0 )
      wire#w1
      I_Contact( "On" )
      "FC300_SetFilm"(Mode := 2, Tiro := "DB215_ProgramData".PhotDelay_Pulses, Prestiro := "DB215_ProgramData".Offset_Pulses, PID := "DB320_PID".PID, SP_Tiro => "Inverter_Data".U241.setpoint, SP_Prestiro => "Inverter_Data".U261.setpoint, Tiro_obiettivo => "DB215_ProgramData".TiroObiettivo)
   END_RUNG
   RUNG wire#powerrail
      I_Contact( "On" )
   END_RUNG wire#w1
   // the same network as SCL:
   IF ("DB08_Prestretch".dbx0_0 OR NOT "On") AND NOT "On" THEN
       "FC300_SetFilm"(Mode := 2,
                       Tiro := "DB215_ProgramData".PhotDelay_Pulses,
                       Prestiro := "DB215_ProgramData".Offset_Pulses,
                       PID := "DB320_PID".PID,
                       SP_Tiro => "Inverter_Data".U241.setpoint,
                       SP_Prestiro => "Inverter_Data".U261.setpoint,
                       Tiro_obiettivo => "DB215_ProgramData".TiroObiettivo);
   END_IF;
END_REGION

REGION Network 17
   RUNG wire#powerrail
      I_Contact( "On" )
      Contact( "On" )
      wire#w1
      Move(in := "CELLA", out1 => "DB322_APP".IN10)
   END_RUNG
   RUNG wire#w1
      Move(in := "DB215_ProgramData".Offset_cella, out1 => "DB322_APP".IN11)
   END_RUNG
   // the same network as SCL:
   IF NOT "On" AND "On" THEN
       "DB322_APP".IN10 := "CELLA";
       "DB322_APP".IN11 := "DB215_ProgramData".Offset_cella;
   END_IF;
END_REGION

REGION Network 18
   // "DB321_PID_M20".PID.M20_P08
   RUNG wire#powerrail
      I_Contact( "On" )
      Contact( "On" )
      wire#w1
      { S7_Templates := "SrcType := DInt"; S7_Expression := "((IN1-IN2)*IN3/IN4)+IN5" } Calculate(in1 := "DB322_APP".IN10, in2 := "DB322_APP".IN11, in3 := 100, in4 := 317, in5 := 58, out => #TempDint)
   END_RUNG
   RUNG wire#w1
      Move(in := #TempDint, out1 => #TempInt)
   END_RUNG
   // the same network as SCL:
   IF NOT "On" AND "On" THEN
       #TempDint := (("DB322_APP".IN10-"DB322_APP".IN11)*100/317)+58;
       #TempInt := #TempDint;
   END_IF;
END_REGION

REGION Network 19
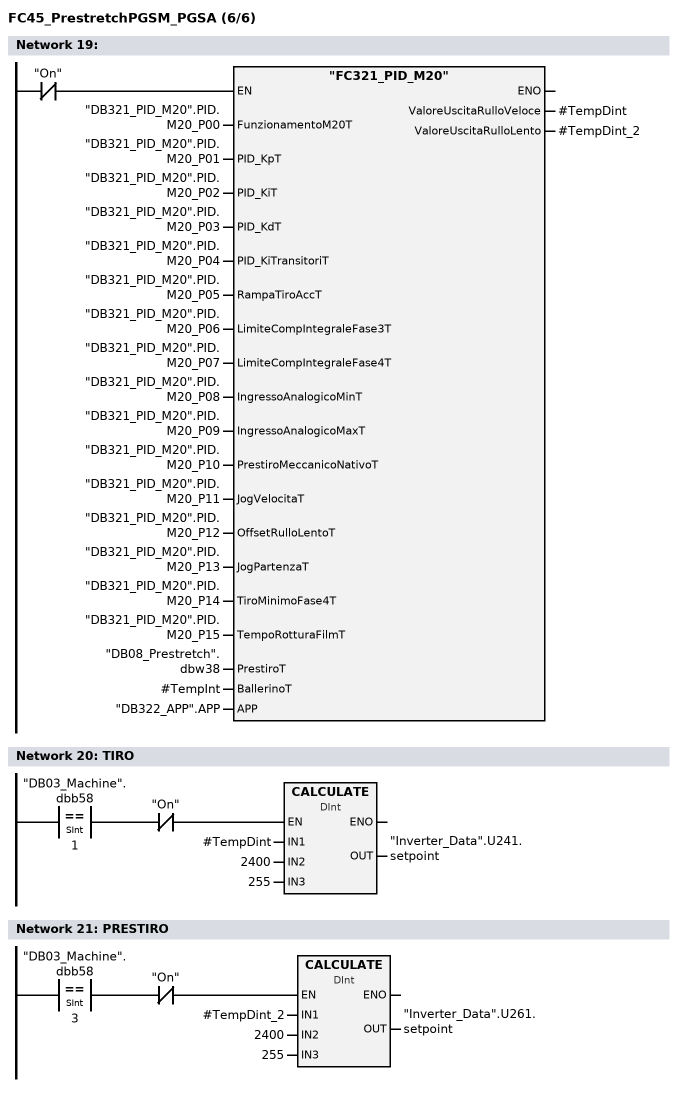
   RUNG wire#powerrail
      I_Contact( "On" )
      "FC321_PID_M20"(FunzionamentoM20T := "DB321_PID_M20".PID.M20_P00, PID_KpT := "DB321_PID_M20".PID.M20_P01, PID_KiT := "DB321_PID_M20".PID.M20_P02, PID_KdT := "DB321_PID_M20".PID.M20_P03, PID_KiTransitoriT := "DB321_PID_M20".PID.M20_P04, RampaTiroAccT := "DB321_PID_M20".PID.M20_P05, LimiteCompIntegraleFase3T := "DB321_PID_M20".PID.M20_P06, LimiteCompIntegraleFase4T := "DB321_PID_M20".PID.M20_P07, IngressoAnalogicoMinT := "DB321_PID_M20".PID.M20_P08, IngressoAnalogicoMaxT := "DB321_PID_M20".PID.M20_P09, PrestiroMeccanicoNativoT := "DB321_PID_M20".PID.M20_P10, JogVelocitaT := "DB321_PID_M20".PID.M20_P11, OffsetRulloLentoT := "DB321_PID_M20".PID.M20_P12, JogPartenzaT := "DB321_PID_M20".PID.M20_P13, TiroMinimoFase4T := "DB321_PID_M20".PID.M20_P14, TempoRotturaFilmT := "DB321_PID_M20".PID.M20_P15, PrestiroT := "DB08_Prestretch".dbw38, BallerinoT := #TempInt, APP := "DB322_APP".APP, ValoreUscitaRulloVeloce => #TempDint, ValoreUscitaRulloLento => #TempDint_2)
   END_RUNG
   // the same network as SCL:
   IF NOT "On" THEN
       "FC321_PID_M20"(FunzionamentoM20T := "DB321_PID_M20".PID.M20_P00,
                       PID_KpT := "DB321_PID_M20".PID.M20_P01,
                       PID_KiT := "DB321_PID_M20".PID.M20_P02,
                       PID_KdT := "DB321_PID_M20".PID.M20_P03,
                       PID_KiTransitoriT := "DB321_PID_M20".PID.M20_P04,
                       RampaTiroAccT := "DB321_PID_M20".PID.M20_P05,
                       LimiteCompIntegraleFase3T := "DB321_PID_M20".PID.M20_P06,
                       LimiteCompIntegraleFase4T := "DB321_PID_M20".PID.M20_P07,
                       IngressoAnalogicoMinT := "DB321_PID_M20".PID.M20_P08,
                       IngressoAnalogicoMaxT := "DB321_PID_M20".PID.M20_P09,
                       PrestiroMeccanicoNativoT := "DB321_PID_M20".PID.M20_P10,
                       JogVelocitaT := "DB321_PID_M20".PID.M20_P11,
                       OffsetRulloLentoT := "DB321_PID_M20".PID.M20_P12,
                       JogPartenzaT := "DB321_PID_M20".PID.M20_P13,
                       TiroMinimoFase4T := "DB321_PID_M20".PID.M20_P14,
                       TempoRotturaFilmT := "DB321_PID_M20".PID.M20_P15,
                       PrestiroT := "DB08_Prestretch".dbw38,
                       BallerinoT := #TempInt,
                       APP := "DB322_APP".APP,
                       ValoreUscitaRulloVeloce => #TempDint,
                       ValoreUscitaRulloLento => #TempDint_2);
   END_IF;
END_REGION

REGION Network 20: TIRO
   RUNG wire#powerrail
      { S7_Templates := "SrcType := SInt" } EQ_Contact(in1 := "DB03_Machine".dbb58, in2 := 1)
      I_Contact( "On" )
      { S7_Templates := "SrcType := DInt"; S7_Expression := "IN1*IN2/IN3" } Calculate(in1 := #TempDint, in2 := 2400, in3 := 255, out => "Inverter_Data".U241.setpoint)
   END_RUNG
   // the same network as SCL:
   IF ("DB03_Machine".dbb58 = 1) AND NOT "On" THEN
       "Inverter_Data".U241.setpoint := #TempDint*2400/255;
   END_IF;
END_REGION

REGION Network 21: PRESTIRO
   RUNG wire#powerrail
      { S7_Templates := "SrcType := SInt" } EQ_Contact(in1 := "DB03_Machine".dbb58, in2 := 3)
      I_Contact( "On" )
      { S7_Templates := "SrcType := DInt"; S7_Expression := "IN1*IN2/IN3" } Calculate(in1 := #TempDint_2, in2 := 2400, in3 := 255, out => "Inverter_Data".U261.setpoint)
   END_RUNG
   // the same network as SCL:
   IF ("DB03_Machine".dbb58 = 3) AND NOT "On" THEN
       "Inverter_Data".U261.setpoint := #TempDint_2*2400/255;
   END_IF;
END_REGION
END_FUNCTION

FUNCTION "FC300_SetFilm" : Void
{ S7_Optimized_Access := 'TRUE' }
VERSION : 0.1
   VAR_INPUT 
      Mode : UInt;
      Tiro : UInt;
      Prestiro : UInt;
   END_VAR

   VAR_OUTPUT 
      SP_Tiro : Real;
      SP_Prestiro : Real;
      Tiro_obiettivo : UInt;
   END_VAR

   VAR_IN_OUT 
      PID : "PID";
   END_VAR

   VAR_TEMP 
      freqT : DInt;
      freqP : DInt;
      tempo : UInt;
      t_temp : Time;
      velocita : DInt;
      correttivoTiro : UInt;
      correttivoPrestiro : UInt;
      rapporto : DInt;
      tiro_temp : UInt;
      clock : Bool;
   END_VAR

   VAR CONSTANT 
      BASE_PRESTIRO : UInt := 100;
      MAX_PRESTIRO_T0 : UInt := 75;
      MAX_PRESTIRO_PVS : UInt := 400;
      RAPP_PRES : UInt := 200;
   END_VAR


BEGIN
	(**)
	
	#freqT := 0;
	#freqP := 0;
	
	//Copia del valore di tiro per confronti in gestione RAMPA [partenza/fine ciclo] (OB30)
	#Tiro_obiettivo := #Tiro;
	
	IF (#PID.setTiro) THEN
	    //Fisso il tiro obiettivo senza passare dalla rampa. Mi serve in avvio ciclo o quando riparto
	    //#PID.tiro := #Tiro;
	    #PID.setTiro := FALSE;
	    //"SetFilmStep" := 1;
	END_IF;
	
	//#tiro_temp := #PID.tiro;
	
	//CARRELLO PVS
	//
	IF (#Mode = 2) THEN //FILM_RUN
	    //Eseguo il calcolo dei parametri (PID) solo ad ogni nuovo valore letto dalla cella (scheda prestiro)
	    IF ("PrestNewValue") THEN
	        "FC320_PID_ParamCalc"(Tiro := #PID.tiro,
	                              Offset_cella := "DB215_ProgramData".Offset_cella,
	                              PID := #PID);
	        "PrestNewValue" := 0;
	    END_IF;
	    //Frequenza TIRO
	    #velocita := #PID.segnale;
	    #freqT := #velocita;
	    (*
	    //Correttivo TIRO
	    #correttivoTiro := (#MAX_PRESTIRO_T0 - 15);//"DB230_Parameters".P_PRESTMIN);
	    #correttivoTiro := (#correttivoTiro * (100 - #Tiro)) / 100;
	    //CorrettivoPRESTIRO
	    #correttivoPrestiro := ((#MAX_PRESTIRO_PVS - #Prestiro) * #Tiro) / 500;
	    //    
	    #rapporto := #BASE_PRESTIRO + #correttivoTiro - #correttivoPrestiro;
	    #rapporto := #rapporto + #Prestiro;
	    #rapporto := #rapporto + 15;//"DB230_Parameters".P_PRESTMIN;
	    //    
	    #velocita := #velocita * #RAPP_PRES;
	    #velocita := #velocita / #rapporto;
	    *)
	    //Frequenza PRESTIRO
	    #rapporto := #BASE_PRESTIRO + #Prestiro;
	    #freqP := #velocita * #RAPP_PRES / #rapporto;
	    //#freqP := #velocita*2/5;
	    //
	    //SP_INVERTER SIEMENS IN RPM (1500@50HZ) -> CONVERSIONE SECONDO PROPORZIONE    
	    #SP_Tiro := DINT_TO_REAL(#freqT * 5);//10);//10);
	    IF (#SP_Tiro >= 3000.0) THEN
	        #SP_Tiro := 3000.0;
	    END_IF;
	    #SP_Prestiro := DINT_TO_REAL(#freqP * 5);//10);//10);
	    IF (#SP_Prestiro >= 3000.0) THEN
	        #SP_Prestiro := 3000.0;
	    END_IF;
	    //
	ELSIF (#Mode = 1) THEN  // FILM_STOP - Freq.Rulli = 0 (per strappare il film durante il taglio)
	    #SP_Tiro := 0;
	    #SP_Prestiro := 0;
	ELSIF (#Mode = 3) THEN     // FILM_MANUAL - Svolgimento film in manuale
	    #SP_Tiro := 1500;
	    #SP_Prestiro := 1500;
	ELSIF (#Mode = 0) THEN    // FILM_DISABLE
	    #SP_Tiro := 0;
	    #SP_Prestiro := 0;
	END_IF;
	//
	(*
	//Film rotto o esaurito
	//
	//IF "CELLA" >= ("DB215_ProgramData".Offset_cella + 10) AND "Timer".T21.Q THEN
	//
	IF "DB230_Parameters".FilmEndEn THEN
	    IF "DB02_Timers".T021.Q THEN
	        "FilmEnd" := 1;
	        "FilmEnd2" := 1;
	    END_IF;
	    IF "DB200_Supervisor".State_Stop = 110 THEN
	        "FilmEnd" := 0;
	    END_IF;
	END_IF;
	*)
END_FUNCTION

FUNCTION "FC320_PID_ParamCalc" : Void
{ S7_Optimized_Access := 'TRUE' }
VERSION : 0.1
   VAR_INPUT 
      Tiro : UInt;
      Offset_cella : Int;
   END_VAR

   VAR_IN_OUT 
      PID : "PID";
   END_VAR

   VAR_TEMP 
      t : UInt;
      errore : DInt;
      setPoint : DInt;
      DIV_P : DInt;
      DIV_I : DInt;
      CELLA_DINT : DInt;
      OFFSET_CELLA_DINT : DInt;
      TEMPDINT : DInt;
   END_VAR


BEGIN
	(**)
	// //rotary
	// //const USHORT #pTiro[11] = {140,120,100,90,80,70,60,50,40,30,20};
	// //const USHORT #iTiro[11] = {140,120,100,90,80,70,60,50,40,30,20};
	// //ROTOTECH3000
	// //const USHORT #pTiro[11] = {70,60,50,45,40,35,30,25,20,20,20};
	// //const USHORT #iTiro[11] = {70,60,50,45,40,35,30,25,20,20,20};
	// //
	// #setPoint := 0;
	// #DIV_P := 200;     //Divisore per comp.proporzionale
	// #DIV_I := 1000;    //Divisore per comp.integrale
	// #OFFSET_CELLA_DINT := INT_TO_DINT(#Offset_cella);
	// //Valori moltiplicativi per proporzionale + integrativo (da vettori)
	// #t:=#Tiro/10;
	// #PID.vParP := "DB215_ProgramData".pTiro[#t];
	// #PID.vParI := "DB215_ProgramData".iTiro[#t];
	// //SET-POINT
	// #setPoint := (#Tiro * "DB230_Parameters".P_DELTA / 10);
	// #setPoint := #setPoint + "DB230_Parameters".P_TIROMIN;
	// //
	// #PID.setPointShow := DINT_TO_UINT(#setPoint + #OFFSET_CELLA_DINT);
	// //    
	// IF (#PID.svuota) THEN
	//     #PID.integrativo := 0;
	//     #PID.svuota := FALSE;
	// END_IF;
	// //
	// //Cella di carico
	// "CELLA" := "MB_REGISTERS".ADDR_08_RD.REG_0;
	// #CELLA_DINT := INT_TO_DINT("CELLA");
	// #CELLA_DINT := #CELLA_DINT - #OFFSET_CELLA_DINT;
	// //
	// //ERRORE: CELLA (feedback) - SETPOINT
	// #errore := ((#CELLA_DINT * UINT_TO_DINT("DB230_Parameters".P_GAIN)) / 100) - #setPoint;
	// //
	// //Gestione componente PROPORZIONALE
	// //
	// IF (#PID.vParP <> 0) THEN
	//     #PID.proporzionale := (#errore * #PID.vParP) / #DIV_P;
	//     IF (#PID.proporzionale < 0) THEN
	//         #PID.proporzionale := 0;
	//     END_IF;
	//     IF (#PID.proporzionale > 1000) THEN
	//         #PID.proporzionale := 1000;
	//     END_IF;
	// ELSE
	//     #PID.proporzionale := 0;
	// END_IF;
	// //
	// #PID.segnale := #PID.proporzionale;
	// //
	// //Gestione componente INTEGRALE
	// //
	// IF (#PID.vParI <> 0) THEN
	//     #errore := (#errore * #PID.vParI) / #DIV_I;
	//     #PID.integrativo := #PID.integrativo + #errore;
	// //    
	//     #PID.integrativo := #PID.integrativo * 998 / 1000; // Rotary 995 (con cella di carico in alto 990)
	// //
	//     IF (#PID.integrativo < 0) THEN
	//         #PID.integrativo := 0;
	//     END_IF;
	//     IF (#PID.integrativo > 1000) THEN
	//         #PID.integrativo := 1000;
	//     END_IF;
	// ELSE
	//     #PID.integrativo := 0;
	// END_IF;
	// //Segnale complessivo "PID"
	// #PID.segnale := #PID.segnale + #PID.integrativo;
	// //Errore
	// "ERR" := #errore;
	// //
	// //rotary
	//const USHORT #pTiro[11] = {140,120,100,90,80,70,60,50,40,30,20};
	//const USHORT #iTiro[11] = {140,120,100,90,80,70,60,50,40,30,20};
	//ROTOTECH3000
	//const USHORT #pTiro[11] = {70,60,50,45,40,35,30,25,20,20,20};
	//const USHORT #iTiro[11] = {70,60,50,45,40,35,30,25,20,20,20};
	//
	//
	#setPoint := 0;
	#DIV_P := 200;     //Divisore per comp.proporzionale
	#DIV_I := 1000;    //Divisore per comp.integrale
	#OFFSET_CELLA_DINT := INT_TO_DINT(#Offset_cella);
	//Valori moltiplicativi per proporzionale + integrativo (da vettori)
	#t := #Tiro / 10;
	#PID.vParP := "DB215_ProgramData".pTiro[#t];
	#PID.vParI := "DB215_ProgramData".iTiro[#t];
	//SET-POINT
	//#setPoint := (#Tiro * "DB230_Parameters".P_DELTA / 10) + "DB230_Parameters".P_TIROMIN + #OFFSET_CELLA_DINT;
	//
	#setPoint := (#Tiro * INT_TO_DINT("DB215_ProgramData".MLC_HeightPulses) / 10) + INT_TO_DINT("DB215_ProgramData".MLC_Rounds) + #OFFSET_CELLA_DINT;
	//
	//
	#PID.setPointShow := DINT_TO_UINT(#setPoint);
	//    
	IF (#PID.svuota) THEN
	    #PID.integrativo := 0;
	    #PID.svuota := FALSE;
	END_IF;
	//
	//Cella di carico
	//"CELLA" := "MB_REGISTERS".ADDR_08_RD.REG_0;
	#CELLA_DINT := INT_TO_DINT("CELLA");
	//#CELLA_DINT := #CELLA_DINT - #OFFSET_CELLA_DINT;
	//
	//ERRORE: CELLA (feedback) - SETPOINT
	//#errore := ((#CELLA_DINT * UINT_TO_DINT("DB230_Parameters".P_GAIN)) / 100) - #setPoint;
	#errore := #CELLA_DINT - #setPoint;
	//
	//Gestione componente PROPORZIONALE
	//
	IF (#PID.vParP <> 0) THEN
	    #PID.proporzionale := (#errore * #PID.vParP) / #DIV_P;
	    IF (#PID.proporzionale < 0) THEN
	        #PID.proporzionale := 0;
	    END_IF;
	    IF (#PID.proporzionale > 1000) THEN
	        #PID.proporzionale := 1000;
	    END_IF;
	ELSE
	    #PID.proporzionale := 0;
	END_IF;
	//
	#PID.segnale := #PID.proporzionale;
	//
	//Gestione componente INTEGRALE
	//
	IF (#PID.vParI <> 0) THEN
	    #errore := (#errore * #PID.vParI) / #DIV_I;
	    #PID.integrativo := #PID.integrativo + #errore;
	    //    
	    #PID.integrativo := #PID.integrativo * 990 / 1000; // Rotary 995 (con cella di carico in alto 990)
	    //
	    IF (#PID.integrativo < 0) THEN
	        #PID.integrativo := 0;
	    END_IF;
	    IF (#PID.integrativo > 1000) THEN
	        #PID.integrativo := 1000;
	    END_IF;
	ELSE
	    #PID.integrativo := 0;
	END_IF;
	//Segnale complessivo "PID"
	#PID.segnale := #PID.segnale + #PID.integrativo;
	//Errore
	"ERR" := #errore;
	//
	(**)
	
END_FUNCTION

FUNCTION "FC63_StretchPGSAoutPWM" : Void   // FC63, LAD
{ S7_Optimized_Access := 'FALSE' }
AUTHOR : PaZan
VERSION : 0.1
// stored: AutoNumber false, IsIECCheckEnabled false, SetENOAutomatically false, UDAEnableTagReadback false
   VAR_TEMP   // added for the SCL form of the ladder/FBD networks
      _w1 : Bool;
   END_VAR
BEGIN

REGION Network 1
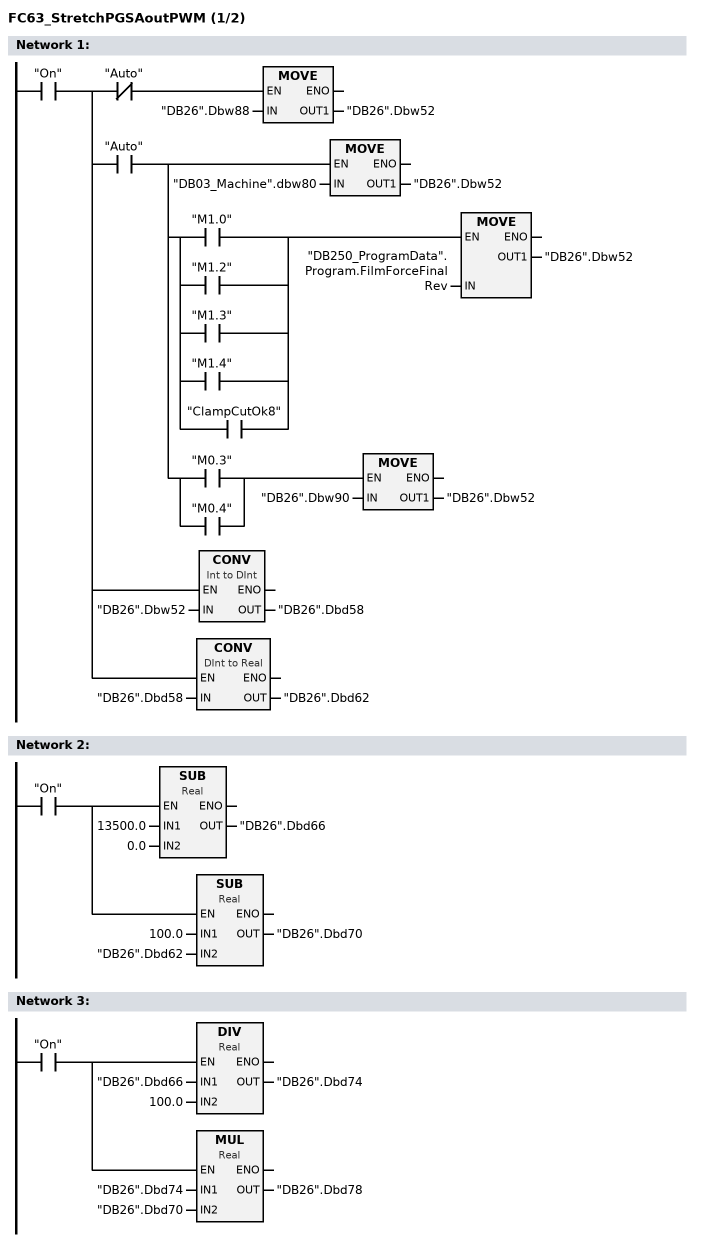
   RUNG wire#powerrail
      Contact( "On" )
      wire#w1
      I_Contact( "Auto" )
      { S7_GenerateENO := "TRUE" } Move(in := "DB26".Dbw88, out1 => "DB26".Dbw52)
   END_RUNG
   RUNG wire#w1
      Contact( "Auto" )
      wire#w2
      { S7_GenerateENO := "TRUE" } Move(in := "DB03_Machine".dbw80, out1 => "DB26".Dbw52)
   END_RUNG
   RUNG wire#w2
      Contact( "M1.0" )
      wire#w3
      { S7_GenerateENO := "TRUE" } Move(in := "DB250_ProgramData".Program.FilmForceFinalRev, out1 => "DB26".Dbw52)
   END_RUNG
   RUNG wire#w2
      Contact( "M1.2" )
   END_RUNG wire#w3
   RUNG wire#w2
      Contact( "M1.3" )
   END_RUNG wire#w3
   RUNG wire#w2
      Contact( "M1.4" )
   END_RUNG wire#w3
   RUNG wire#w2
      Contact( "ClampCutOk8" )
   END_RUNG wire#w3
   RUNG wire#w2
      Contact( "M0.3" )
      wire#w4
      { S7_GenerateENO := "TRUE" } Move(in := "DB26".Dbw90, out1 => "DB26".Dbw52)
   END_RUNG
   RUNG wire#w2
      Contact( "M0.4" )
   END_RUNG wire#w4
   RUNG wire#w1
      { S7_Templates := "[SrcType := Int, DestType := DInt]"; S7_GenerateENO := "TRUE" } Convert(in := "DB26".Dbw52, out => "DB26".Dbd58)
   END_RUNG
   RUNG wire#w1
      { S7_Templates := "[SrcType := DInt, DestType := Real]"; S7_GenerateENO := "TRUE" } Convert(in := "DB26".Dbd58, out => "DB26".Dbd62)
   END_RUNG
   // the same network as SCL:
   IF "On" AND NOT "Auto" THEN "DB26".Dbw52 := "DB26".Dbw88; END_IF;
   #_w1 := "On" AND "Auto";
   IF #_w1 THEN "DB26".Dbw52 := "DB03_Machine".dbw80; END_IF;
   IF #_w1 AND ("M1.0" OR "M1.2" OR "M1.3" OR "M1.4" OR "ClampCutOk8") THEN
       "DB26".Dbw52 := "DB250_ProgramData".Program.FilmForceFinalRev;
   END_IF;
   IF #_w1 AND ("M0.3" OR "M0.4") THEN "DB26".Dbw52 := "DB26".Dbw90; END_IF;
   IF "On" THEN
       "DB26".Dbd58 := INT_TO_DINT("DB26".Dbw52);
       "DB26".Dbd62 := DINT_TO_REAL("DB26".Dbd58);
   END_IF;
END_REGION

REGION Network 2
   RUNG wire#powerrail
      Contact( "On" )
      wire#w1
      { S7_Templates := "SrcType := Real"; S7_GenerateENO := "TRUE" } Sub(in1 := 13500.0, in2 := 0.0, out => "DB26".Dbd66)
   END_RUNG
   RUNG wire#w1
      { S7_Templates := "SrcType := Real"; S7_GenerateENO := "TRUE" } Sub(in1 := 100.0, in2 := "DB26".Dbd62, out => "DB26".Dbd70)
   END_RUNG
   // the same network as SCL:
   IF "On" THEN
       "DB26".Dbd66 := 13500.0 - 0.0;
       "DB26".Dbd70 := 100.0 - "DB26".Dbd62;
   END_IF;
END_REGION

REGION Network 3
   RUNG wire#powerrail
      Contact( "On" )
      wire#w1
      { S7_Templates := "SrcType := Real"; S7_GenerateENO := "TRUE" } Div(in1 := "DB26".Dbd66, in2 := 100.0, out => "DB26".Dbd74)
   END_RUNG
   RUNG wire#w1
      { S7_Templates := "SrcType := Real"; S7_GenerateENO := "TRUE" } Mul(in1 := "DB26".Dbd74, in2 := "DB26".Dbd70, out => "DB26".Dbd78)
   END_RUNG
   // the same network as SCL:
   IF "On" THEN
       "DB26".Dbd74 := "DB26".Dbd66 / 100.0;
       "DB26".Dbd78 := "DB26".Dbd74 * "DB26".Dbd70;
   END_IF;
END_REGION

REGION Network 4: Trunc and copy value for stretch torque in analogic out
   // PAW130
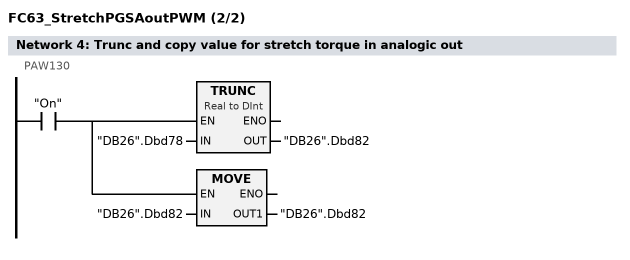
   RUNG wire#powerrail
      Contact( "On" )
      wire#w1
      { S7_Templates := "[SrcType := Real, DestType := DInt]"; S7_GenerateENO := "TRUE" } Trunc(in := "DB26".Dbd78, out => "DB26".Dbd82)
   END_RUNG
   RUNG wire#w1
      { S7_GenerateENO := "TRUE" } Move(in := "DB26".Dbd82, out1 => "DB26".Dbd82)
   END_RUNG
   // the same network as SCL:
   IF "On" THEN
       "DB26".Dbd82 := TRUNC("DB26".Dbd78);
       "DB26".Dbd82 := "DB26".Dbd82;
   END_IF;
END_REGION
END_FUNCTION

FUNCTION "FC77_Conveyor_1_IN_1_OUT" : Void   // FC77, LAD
TITLE = Conveyor_1_IN_1_OUT
{ S7_Optimized_Access := 'TRUE' }
VERSION : 0.1
// stored: AutoNumber false, IsIECCheckEnabled false, SetENOAutomatically false, UDAEnableTagReadback false
   VAR_TEMP   // added for the SCL form of the ladder/FBD networks
      _w1 : Bool;
   END_VAR
BEGIN

REGION Network 1: Manual operation for conveyor
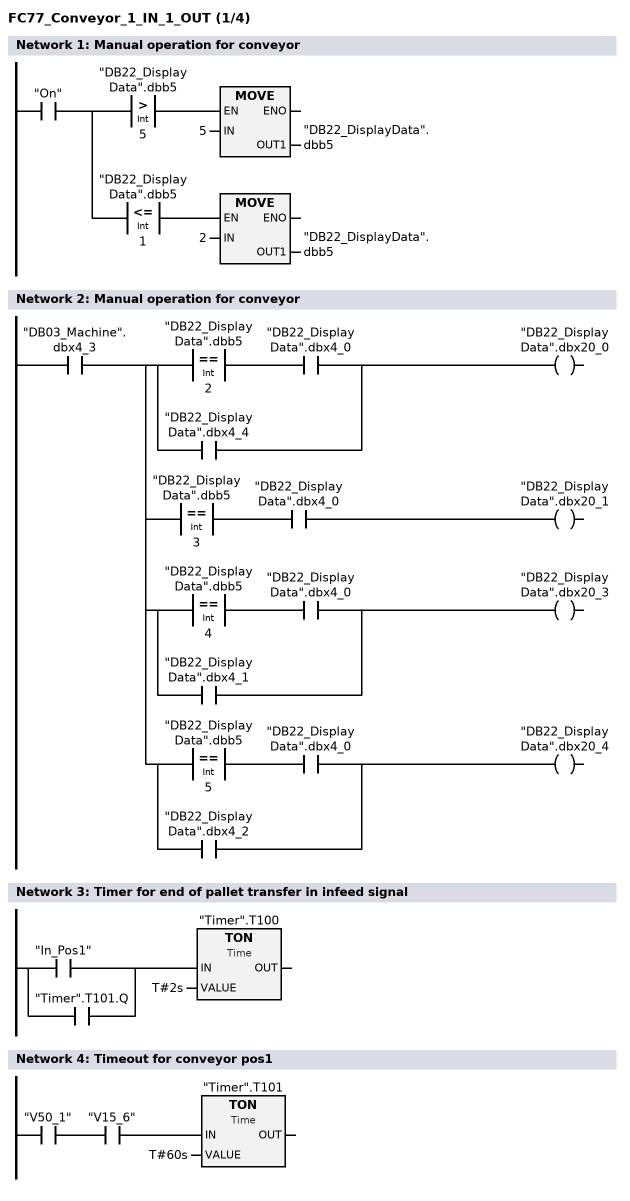
   RUNG wire#powerrail
      Contact( "On" )
      wire#w1
      { S7_Templates := "SrcType := Int" } GT_Contact(in1 := "DB22_DisplayData".dbb5, in2 := 5)
      { S7_GenerateENO := "TRUE" } Move(in := 5, out1 => "DB22_DisplayData".dbb5)
   END_RUNG
   RUNG wire#w1
      { S7_Templates := "SrcType := Int" } LE_Contact(in1 := "DB22_DisplayData".dbb5, in2 := 1)
      { S7_GenerateENO := "TRUE" } Move(in := 2, out1 => "DB22_DisplayData".dbb5)
   END_RUNG
   // the same network as SCL:
   IF "On" AND ("DB22_DisplayData".dbb5 > 5) THEN "DB22_DisplayData".dbb5 := 5; END_IF;
   IF "On" AND ("DB22_DisplayData".dbb5 <= 1) THEN "DB22_DisplayData".dbb5 := 2; END_IF;
END_REGION

REGION Network 2: Manual operation for conveyor
   RUNG wire#powerrail
      Contact( "DB03_Machine".dbx4_3 )
      wire#w1
      { S7_Templates := "SrcType := Int" } EQ_Contact(in1 := "DB22_DisplayData".dbb5, in2 := 2)
      Contact( "DB22_DisplayData".dbx4_0 )
      wire#w2
      Coil( "DB22_DisplayData".dbx20_0 )
   END_RUNG
   RUNG wire#w1
      Contact( "DB22_DisplayData".dbx4_4 )
   END_RUNG wire#w2
   RUNG wire#w1
      { S7_Templates := "SrcType := Int" } EQ_Contact(in1 := "DB22_DisplayData".dbb5, in2 := 3)
      Contact( "DB22_DisplayData".dbx4_0 )
      Coil( "DB22_DisplayData".dbx20_1 )
   END_RUNG
   RUNG wire#w1
      { S7_Templates := "SrcType := Int" } EQ_Contact(in1 := "DB22_DisplayData".dbb5, in2 := 4)
      Contact( "DB22_DisplayData".dbx4_0 )
      wire#w3
      Coil( "DB22_DisplayData".dbx20_3 )
   END_RUNG
   RUNG wire#w1
      Contact( "DB22_DisplayData".dbx4_1 )
   END_RUNG wire#w3
   RUNG wire#w1
      { S7_Templates := "SrcType := Int" } EQ_Contact(in1 := "DB22_DisplayData".dbb5, in2 := 5)
      Contact( "DB22_DisplayData".dbx4_0 )
      wire#w4
      Coil( "DB22_DisplayData".dbx20_4 )
   END_RUNG
   RUNG wire#w1
      Contact( "DB22_DisplayData".dbx4_2 )
   END_RUNG wire#w4
   // the same network as SCL:
   "DB22_DisplayData".dbx20_0 := "DB03_Machine".dbx4_3 AND ((("DB22_DisplayData".dbb5 = 2) AND "DB22_DisplayData".dbx4_0) OR "DB22_DisplayData".dbx4_4);
   "DB22_DisplayData".dbx20_1 := "DB03_Machine".dbx4_3 AND ("DB22_DisplayData".dbb5 = 3) AND "DB22_DisplayData".dbx4_0;
   "DB22_DisplayData".dbx20_3 := "DB03_Machine".dbx4_3 AND ((("DB22_DisplayData".dbb5 = 4) AND "DB22_DisplayData".dbx4_0) OR "DB22_DisplayData".dbx4_1);
   "DB22_DisplayData".dbx20_4 := "DB03_Machine".dbx4_3 AND ((("DB22_DisplayData".dbb5 = 5) AND "DB22_DisplayData".dbx4_0) OR "DB22_DisplayData".dbx4_2);
END_REGION

REGION Network 3: Timer for end of pallet transfer in infeed signal
   "Timer".T100.TON(IN := "In_Pos1" OR "Timer".T101.Q, PT := T#2s);   // TON coil
END_REGION

REGION Network 4: Timeout for conveyor pos1
   "Timer".T101.TON(IN := "V50_1" AND "V15_6", PT := T#60s);   // TON coil
END_REGION

REGION Network 5: Time to load with forklift
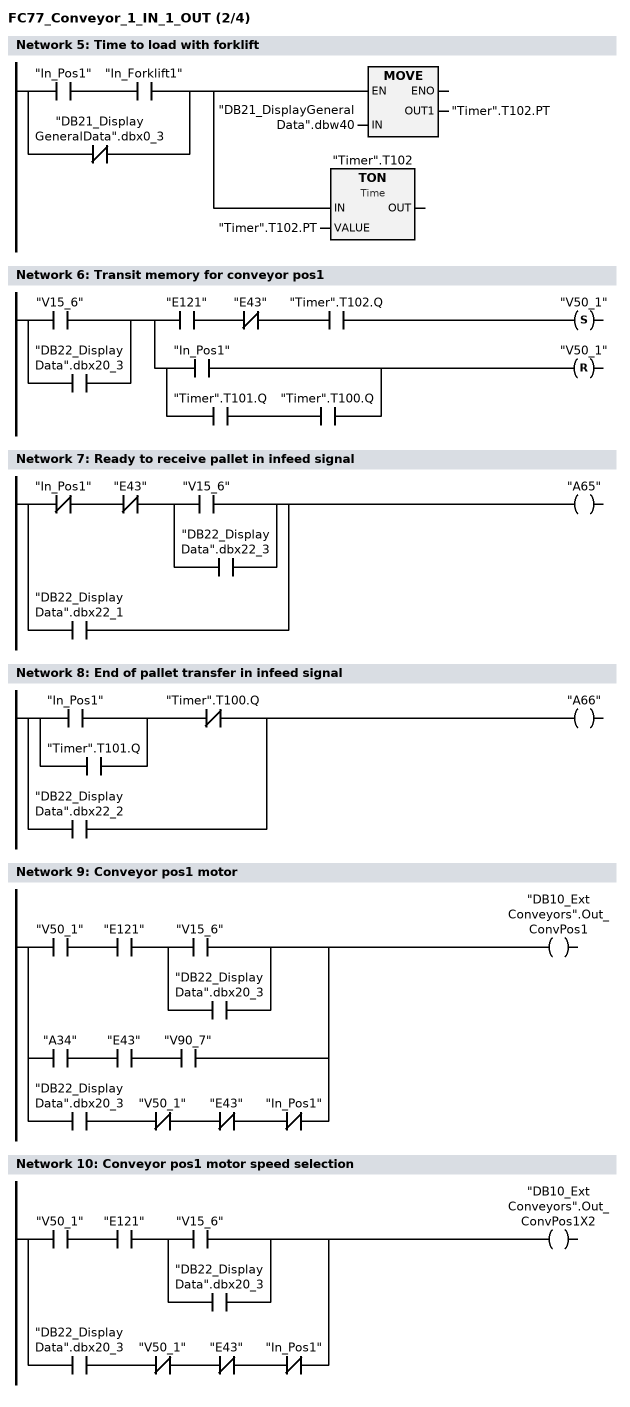
   #_w1 := ("In_Pos1" AND "In_Forklift1") OR NOT "DB21_DisplayGeneralData".dbx0_3;
   IF #_w1 THEN "Timer".T102.PT := "DB21_DisplayGeneralData".dbw40; END_IF;
   "Timer".T102.TON(IN := #_w1, PT := "Timer".T102.PT);   // TON coil
END_REGION

REGION Network 6: Transit memory for conveyor pos1
   RUNG wire#powerrail
      Contact( "V15_6" )
      wire#w1
      Contact( "E121" )
      I_Contact( "E43" )
      Contact( "Timer".T102.Q )
      S_Coil( "V50_1" )
   END_RUNG
   RUNG wire#powerrail
      Contact( "DB22_DisplayData".dbx20_3 )
   END_RUNG wire#w1
   RUNG wire#w1
      Contact( "In_Pos1" )
      wire#w2
      R_Coil( "V50_1" )
   END_RUNG
   RUNG wire#w1
      Contact( "Timer".T101.Q )
      Contact( "Timer".T100.Q )
   END_RUNG wire#w2
   // the same network as SCL:
   #_w1 := "V15_6" OR "DB22_DisplayData".dbx20_3;
   IF #_w1 AND "E121" AND NOT "E43" AND "Timer".T102.Q THEN "V50_1" := TRUE; END_IF;
   IF #_w1 AND ("In_Pos1" OR ("Timer".T101.Q AND "Timer".T100.Q)) THEN "V50_1" := FALSE; END_IF;
END_REGION

REGION Network 7: Ready to receive pallet in infeed signal
   RUNG wire#powerrail
      I_Contact( "In_Pos1" )
      I_Contact( "E43" )
      wire#w1
      Contact( "V15_6" )
      wire#w2
      Coil( "A65" )
   END_RUNG
   RUNG wire#w1
      Contact( "DB22_DisplayData".dbx22_3 )
   END_RUNG wire#w2
   RUNG wire#powerrail
      Contact( "DB22_DisplayData".dbx22_1 )
   END_RUNG wire#w2
   // the same network as SCL:
   "A65" := (NOT "In_Pos1" AND NOT "E43" AND ("V15_6" OR "DB22_DisplayData".dbx22_3)) OR "DB22_DisplayData".dbx22_1;
END_REGION

REGION Network 8: End of pallet transfer in infeed signal
   RUNG wire#powerrail
      Contact( "In_Pos1" )
      wire#w1
      I_Contact( "Timer".T100.Q )
      wire#w2
      Coil( "A66" )
   END_RUNG
   RUNG wire#powerrail
      Contact( "Timer".T101.Q )
   END_RUNG wire#w1
   RUNG wire#powerrail
      Contact( "DB22_DisplayData".dbx22_2 )
   END_RUNG wire#w2
   // the same network as SCL:
   "A66" := (("In_Pos1" OR "Timer".T101.Q) AND NOT "Timer".T100.Q) OR "DB22_DisplayData".dbx22_2;
END_REGION

REGION Network 9: Conveyor pos1 motor
   RUNG wire#powerrail
      Contact( "V50_1" )
      Contact( "E121" )
      wire#w1
      Contact( "V15_6" )
      wire#w2
      Coil( "DB10_ExtConveyors".Out_ConvPos1 )
   END_RUNG
   RUNG wire#w1
      Contact( "DB22_DisplayData".dbx20_3 )
   END_RUNG wire#w2
   RUNG wire#powerrail
      Contact( "A34" )
      Contact( "E43" )
      Contact( "V90_7" )
   END_RUNG wire#w2
   RUNG wire#powerrail
      Contact( "DB22_DisplayData".dbx20_3 )
      I_Contact( "V50_1" )
      I_Contact( "E43" )
      I_Contact( "In_Pos1" )
   END_RUNG wire#w2
   // the same network as SCL:
   "DB10_ExtConveyors".Out_ConvPos1 := ("V50_1" AND "E121" AND ("V15_6" OR "DB22_DisplayData".dbx20_3)) OR ("A34" AND "E43" AND "V90_7") OR ("DB22_DisplayData".dbx20_3 AND NOT "V50_1" AND NOT "E43" AND NOT "In_Pos1");
END_REGION

REGION Network 10: Conveyor pos1 motor speed selection
   RUNG wire#powerrail
      Contact( "V50_1" )
      Contact( "E121" )
      wire#w1
      Contact( "V15_6" )
      wire#w2
      Coil( "DB10_ExtConveyors".Out_ConvPos1X2 )
   END_RUNG
   RUNG wire#w1
      Contact( "DB22_DisplayData".dbx20_3 )
   END_RUNG wire#w2
   RUNG wire#powerrail
      Contact( "DB22_DisplayData".dbx20_3 )
      I_Contact( "V50_1" )
      I_Contact( "E43" )
      I_Contact( "In_Pos1" )
   END_RUNG wire#w2
   // the same network as SCL:
   "DB10_ExtConveyors".Out_ConvPos1X2 := ("V50_1" AND "E121" AND ("V15_6" OR "DB22_DisplayData".dbx20_3)) OR ("DB22_DisplayData".dbx20_3 AND NOT "V50_1" AND NOT "E43" AND NOT "In_Pos1");
END_REGION

REGION Network 11: Pallet ready in infeed signal (Std signal)
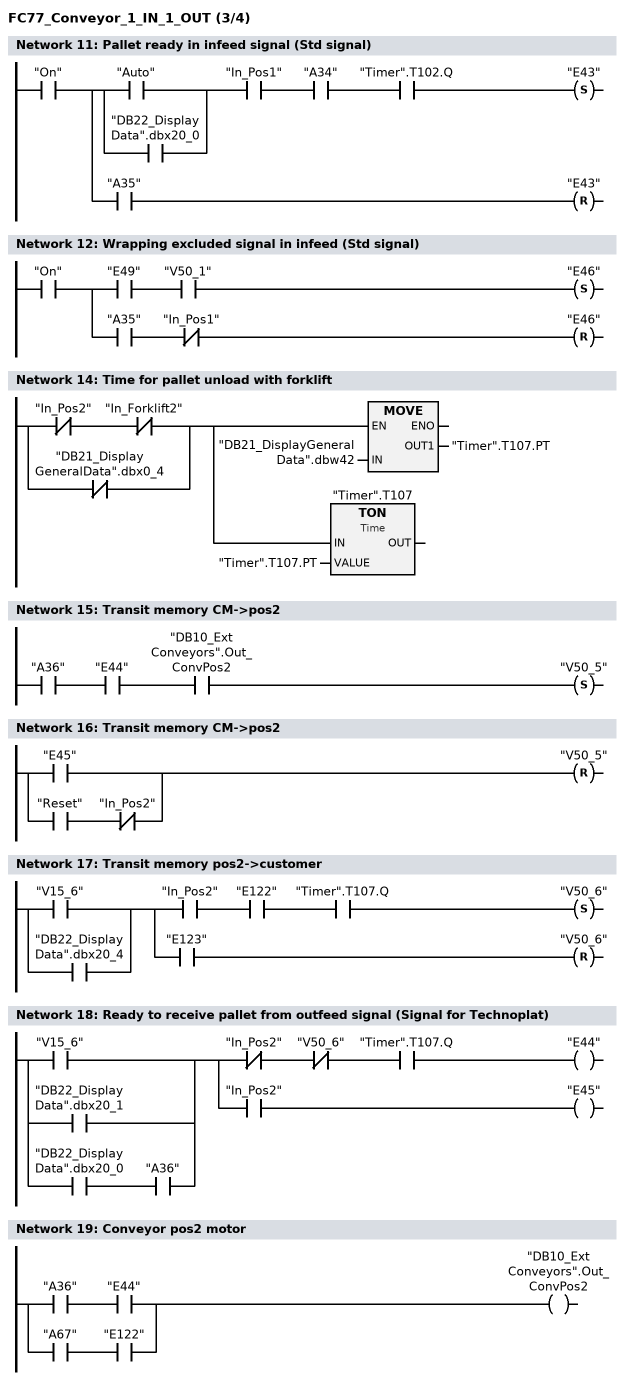
   RUNG wire#powerrail
      Contact( "On" )
      wire#w1
      Contact( "Auto" )
      wire#w2
      Contact( "In_Pos1" )
      Contact( "A34" )
      Contact( "Timer".T102.Q )
      S_Coil( "E43" )
   END_RUNG
   RUNG wire#w1
      Contact( "DB22_DisplayData".dbx20_0 )
   END_RUNG wire#w2
   RUNG wire#w1
      Contact( "A35" )
      R_Coil( "E43" )
   END_RUNG
   // the same network as SCL:
   IF "On" AND ("Auto" OR "DB22_DisplayData".dbx20_0) AND "In_Pos1" AND "A34" AND "Timer".T102.Q THEN
       "E43" := TRUE;
   END_IF;
   IF "On" AND "A35" THEN "E43" := FALSE; END_IF;
END_REGION

REGION Network 12: Wrapping excluded signal in infeed (Std signal)
   RUNG wire#powerrail
      Contact( "On" )
      wire#w1
      Contact( "E49" )
      Contact( "V50_1" )
      S_Coil( "E46" )
   END_RUNG
   RUNG wire#w1
      Contact( "A35" )
      I_Contact( "In_Pos1" )
      R_Coil( "E46" )
   END_RUNG
   // the same network as SCL:
   IF "On" AND "E49" AND "V50_1" THEN "E46" := TRUE; END_IF;
   IF "On" AND "A35" AND NOT "In_Pos1" THEN "E46" := FALSE; END_IF;
END_REGION

REGION Network 13: >>>>>>> OUTFEED CONVEYOR <<<<<<<<
END_REGION

REGION Network 14: Time for pallet unload with forklift
   #_w1 := (NOT "In_Pos2" AND NOT "In_Forklift2") OR NOT "DB21_DisplayGeneralData".dbx0_4;
   IF #_w1 THEN "Timer".T107.PT := "DB21_DisplayGeneralData".dbw42; END_IF;
   "Timer".T107.TON(IN := #_w1, PT := "Timer".T107.PT);   // TON coil
END_REGION

REGION Network 15: Transit memory CM->pos2
   RUNG wire#powerrail
      Contact( "A36" )
      Contact( "E44" )
      Contact( "DB10_ExtConveyors".Out_ConvPos2 )
      S_Coil( "V50_5" )
   END_RUNG
   // the same network as SCL:
   IF "A36" AND "E44" AND "DB10_ExtConveyors".Out_ConvPos2 THEN "V50_5" := TRUE; END_IF;
END_REGION

REGION Network 16: Transit memory CM->pos2
   RUNG wire#powerrail
      Contact( "E45" )
      wire#w1
      R_Coil( "V50_5" )
   END_RUNG
   RUNG wire#powerrail
      Contact( "Reset" )
      I_Contact( "In_Pos2" )
   END_RUNG wire#w1
   // the same network as SCL:
   IF "E45" OR ("Reset" AND NOT "In_Pos2") THEN "V50_5" := FALSE; END_IF;
END_REGION

REGION Network 17: Transit memory pos2->customer
   RUNG wire#powerrail
      Contact( "V15_6" )
      wire#w1
      Contact( "In_Pos2" )
      Contact( "E122" )
      Contact( "Timer".T107.Q )
      S_Coil( "V50_6" )
   END_RUNG
   RUNG wire#powerrail
      Contact( "DB22_DisplayData".dbx20_4 )
   END_RUNG wire#w1
   RUNG wire#w1
      Contact( "E123" )
      R_Coil( "V50_6" )
   END_RUNG
   // the same network as SCL:
   #_w1 := "V15_6" OR "DB22_DisplayData".dbx20_4;
   IF #_w1 AND "In_Pos2" AND "E122" AND "Timer".T107.Q THEN "V50_6" := TRUE; END_IF;
   IF #_w1 AND "E123" THEN "V50_6" := FALSE; END_IF;
END_REGION

REGION Network 18: Ready to receive pallet from outfeed signal (Signal for Technoplat)
   RUNG wire#powerrail
      Contact( "V15_6" )
      wire#w1
      I_Contact( "In_Pos2" )
      I_Contact( "V50_6" )
      Contact( "Timer".T107.Q )
      Coil( "E44" )
   END_RUNG
   RUNG wire#powerrail
      Contact( "DB22_DisplayData".dbx20_1 )
   END_RUNG wire#w1
   RUNG wire#powerrail
      Contact( "DB22_DisplayData".dbx20_0 )
      Contact( "A36" )
   END_RUNG wire#w1
   RUNG wire#w1
      Contact( "In_Pos2" )
      Coil( "E45" )
   END_RUNG
   // the same network as SCL:
   #_w1 := "V15_6" OR "DB22_DisplayData".dbx20_1 OR ("DB22_DisplayData".dbx20_0 AND "A36");
   "E44" := #_w1 AND NOT "In_Pos2" AND NOT "V50_6" AND "Timer".T107.Q;
   "E45" := #_w1 AND "In_Pos2";
END_REGION

REGION Network 19: Conveyor pos2 motor
   RUNG wire#powerrail
      Contact( "A36" )
      Contact( "E44" )
      wire#w1
      Coil( "DB10_ExtConveyors".Out_ConvPos2 )
   END_RUNG
   RUNG wire#powerrail
      Contact( "A67" )
      Contact( "E122" )
   END_RUNG wire#w1
   // the same network as SCL:
   "DB10_ExtConveyors".Out_ConvPos2 := ("A36" AND "E44") OR ("A67" AND "E122");
END_REGION

REGION Network 20: Conveyor pos2 motor speed selection
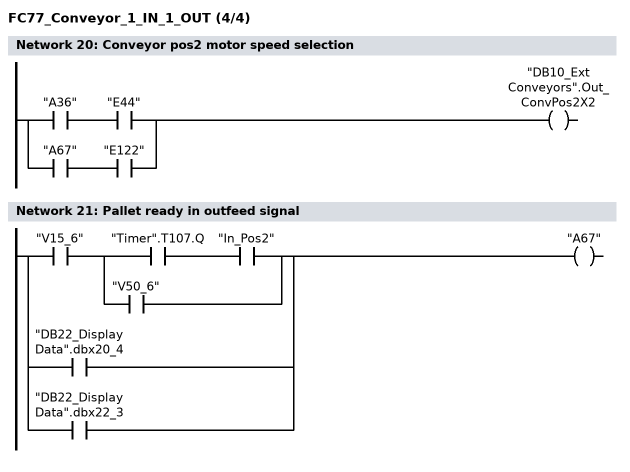
   RUNG wire#powerrail
      Contact( "A36" )
      Contact( "E44" )
      wire#w1
      Coil( "DB10_ExtConveyors".Out_ConvPos2X2 )
   END_RUNG
   RUNG wire#powerrail
      Contact( "A67" )
      Contact( "E122" )
   END_RUNG wire#w1
   // the same network as SCL:
   "DB10_ExtConveyors".Out_ConvPos2X2 := ("A36" AND "E44") OR ("A67" AND "E122");
END_REGION

REGION Network 21: Pallet ready in outfeed signal
   RUNG wire#powerrail
      Contact( "V15_6" )
      wire#w1
      Contact( "Timer".T107.Q )
      Contact( "In_Pos2" )
      wire#w2
      Coil( "A67" )
   END_RUNG
   RUNG wire#w1
      Contact( "V50_6" )
   END_RUNG wire#w2
   RUNG wire#powerrail
      Contact( "DB22_DisplayData".dbx20_4 )
   END_RUNG wire#w2
   RUNG wire#powerrail
      Contact( "DB22_DisplayData".dbx22_3 )
   END_RUNG wire#w2
   // the same network as SCL:
   "A67" := ("V15_6" AND (("Timer".T107.Q AND "In_Pos2") OR "V50_6")) OR "DB22_DisplayData".dbx20_4 OR "DB22_DisplayData".dbx22_3;
END_REGION
END_FUNCTION

FUNCTION "FC78_Conveyor_1_IN_1_OUT_REVERSE" : Void   // FC78, LAD
TITLE = Conveyor_1_IN_1_OUT
{ S7_Optimized_Access := 'TRUE' }
VERSION : 0.1
// stored: AutoNumber false, IsIECCheckEnabled false, SetENOAutomatically false, UDAEnableTagReadback false
   VAR_TEMP   // added for the SCL form of the ladder/FBD networks
      _w1 : Bool;
   END_VAR
BEGIN

REGION Network 1: Manual operation for conveyor
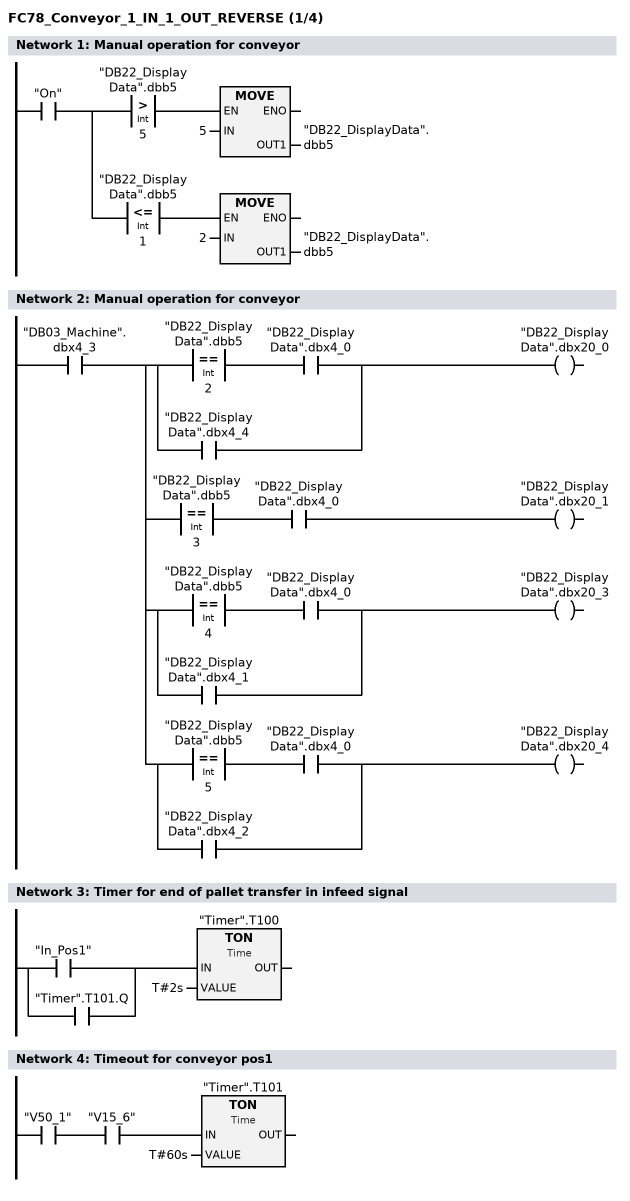
   RUNG wire#powerrail
      Contact( "On" )
      wire#w1
      { S7_Templates := "SrcType := Int" } GT_Contact(in1 := "DB22_DisplayData".dbb5, in2 := 5)
      { S7_GenerateENO := "TRUE" } Move(in := 5, out1 => "DB22_DisplayData".dbb5)
   END_RUNG
   RUNG wire#w1
      { S7_Templates := "SrcType := Int" } LE_Contact(in1 := "DB22_DisplayData".dbb5, in2 := 1)
      { S7_GenerateENO := "TRUE" } Move(in := 2, out1 => "DB22_DisplayData".dbb5)
   END_RUNG
   // the same network as SCL:
   IF "On" AND ("DB22_DisplayData".dbb5 > 5) THEN "DB22_DisplayData".dbb5 := 5; END_IF;
   IF "On" AND ("DB22_DisplayData".dbb5 <= 1) THEN "DB22_DisplayData".dbb5 := 2; END_IF;
END_REGION

REGION Network 2: Manual operation for conveyor
   RUNG wire#powerrail
      Contact( "DB03_Machine".dbx4_3 )
      wire#w1
      { S7_Templates := "SrcType := Int" } EQ_Contact(in1 := "DB22_DisplayData".dbb5, in2 := 2)
      Contact( "DB22_DisplayData".dbx4_0 )
      wire#w2
      Coil( "DB22_DisplayData".dbx20_0 )
   END_RUNG
   RUNG wire#w1
      Contact( "DB22_DisplayData".dbx4_4 )
   END_RUNG wire#w2
   RUNG wire#w1
      { S7_Templates := "SrcType := Int" } EQ_Contact(in1 := "DB22_DisplayData".dbb5, in2 := 3)
      Contact( "DB22_DisplayData".dbx4_0 )
      Coil( "DB22_DisplayData".dbx20_1 )
   END_RUNG
   RUNG wire#w1
      { S7_Templates := "SrcType := Int" } EQ_Contact(in1 := "DB22_DisplayData".dbb5, in2 := 4)
      Contact( "DB22_DisplayData".dbx4_0 )
      wire#w3
      Coil( "DB22_DisplayData".dbx20_3 )
   END_RUNG
   RUNG wire#w1
      Contact( "DB22_DisplayData".dbx4_1 )
   END_RUNG wire#w3
   RUNG wire#w1
      { S7_Templates := "SrcType := Int" } EQ_Contact(in1 := "DB22_DisplayData".dbb5, in2 := 5)
      Contact( "DB22_DisplayData".dbx4_0 )
      wire#w4
      Coil( "DB22_DisplayData".dbx20_4 )
   END_RUNG
   RUNG wire#w1
      Contact( "DB22_DisplayData".dbx4_2 )
   END_RUNG wire#w4
   // the same network as SCL:
   "DB22_DisplayData".dbx20_0 := "DB03_Machine".dbx4_3 AND ((("DB22_DisplayData".dbb5 = 2) AND "DB22_DisplayData".dbx4_0) OR "DB22_DisplayData".dbx4_4);
   "DB22_DisplayData".dbx20_1 := "DB03_Machine".dbx4_3 AND ("DB22_DisplayData".dbb5 = 3) AND "DB22_DisplayData".dbx4_0;
   "DB22_DisplayData".dbx20_3 := "DB03_Machine".dbx4_3 AND ((("DB22_DisplayData".dbb5 = 4) AND "DB22_DisplayData".dbx4_0) OR "DB22_DisplayData".dbx4_1);
   "DB22_DisplayData".dbx20_4 := "DB03_Machine".dbx4_3 AND ((("DB22_DisplayData".dbb5 = 5) AND "DB22_DisplayData".dbx4_0) OR "DB22_DisplayData".dbx4_2);
END_REGION

REGION Network 3: Timer for end of pallet transfer in infeed signal
   "Timer".T100.TON(IN := "In_Pos1" OR "Timer".T101.Q, PT := T#2s);   // TON coil
END_REGION

REGION Network 4: Timeout for conveyor pos1
   "Timer".T101.TON(IN := "V50_1" AND "V15_6", PT := T#60s);   // TON coil
END_REGION

REGION Network 5: Time to load with forklift
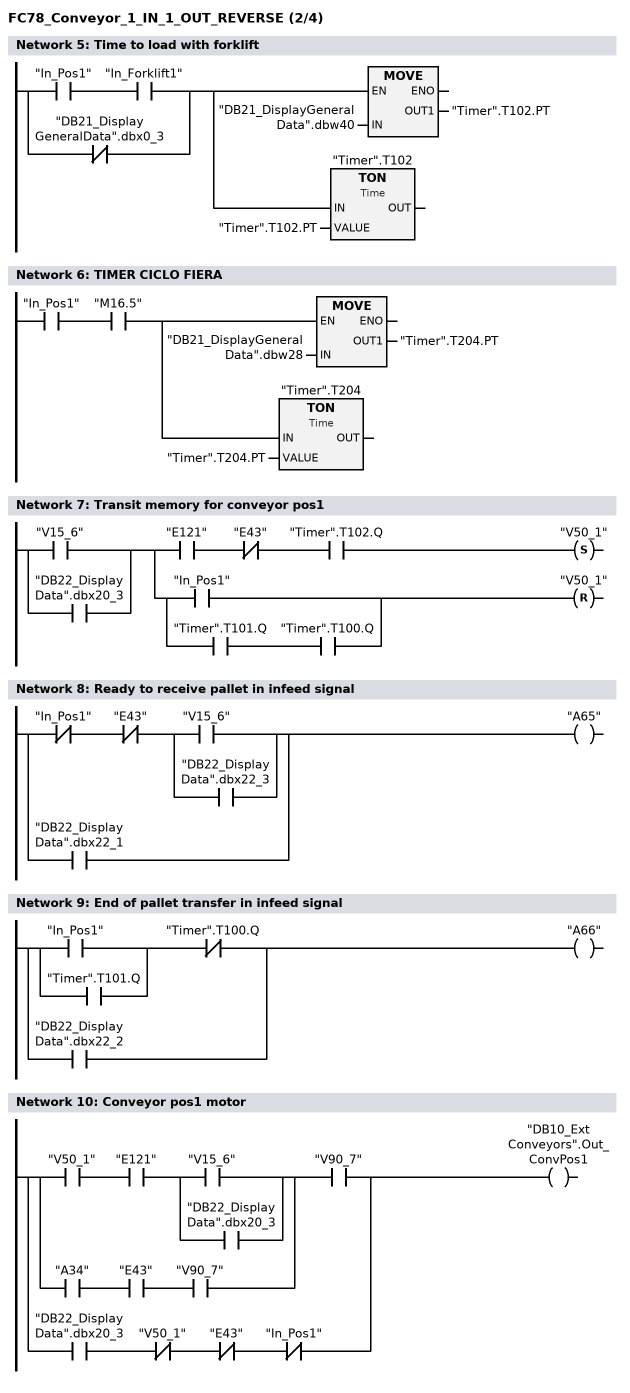
   #_w1 := ("In_Pos1" AND "In_Forklift1") OR NOT "DB21_DisplayGeneralData".dbx0_3;
   IF #_w1 THEN "Timer".T102.PT := "DB21_DisplayGeneralData".dbw40; END_IF;
   "Timer".T102.TON(IN := #_w1, PT := "Timer".T102.PT);   // TON coil
END_REGION

REGION Network 6: TIMER CICLO FIERA
   #_w1 := "In_Pos1" AND "M16.5";
   IF #_w1 THEN "Timer".T204.PT := "DB21_DisplayGeneralData".dbw28; END_IF;
   "Timer".T204.TON(IN := #_w1, PT := "Timer".T204.PT);   // TON coil
END_REGION

REGION Network 7: Transit memory for conveyor pos1
   RUNG wire#powerrail
      Contact( "V15_6" )
      wire#w1
      Contact( "E121" )
      I_Contact( "E43" )
      Contact( "Timer".T102.Q )
      S_Coil( "V50_1" )
   END_RUNG
   RUNG wire#powerrail
      Contact( "DB22_DisplayData".dbx20_3 )
   END_RUNG wire#w1
   RUNG wire#w1
      Contact( "In_Pos1" )
      wire#w2
      R_Coil( "V50_1" )
   END_RUNG
   RUNG wire#w1
      Contact( "Timer".T101.Q )
      Contact( "Timer".T100.Q )
   END_RUNG wire#w2
   // the same network as SCL:
   #_w1 := "V15_6" OR "DB22_DisplayData".dbx20_3;
   IF #_w1 AND "E121" AND NOT "E43" AND "Timer".T102.Q THEN "V50_1" := TRUE; END_IF;
   IF #_w1 AND ("In_Pos1" OR ("Timer".T101.Q AND "Timer".T100.Q)) THEN "V50_1" := FALSE; END_IF;
END_REGION

REGION Network 8: Ready to receive pallet in infeed signal
   RUNG wire#powerrail
      I_Contact( "In_Pos1" )
      I_Contact( "E43" )
      wire#w1
      Contact( "V15_6" )
      wire#w2
      Coil( "A65" )
   END_RUNG
   RUNG wire#w1
      Contact( "DB22_DisplayData".dbx22_3 )
   END_RUNG wire#w2
   RUNG wire#powerrail
      Contact( "DB22_DisplayData".dbx22_1 )
   END_RUNG wire#w2
   // the same network as SCL:
   "A65" := (NOT "In_Pos1" AND NOT "E43" AND ("V15_6" OR "DB22_DisplayData".dbx22_3)) OR "DB22_DisplayData".dbx22_1;
END_REGION

REGION Network 9: End of pallet transfer in infeed signal
   RUNG wire#powerrail
      Contact( "In_Pos1" )
      wire#w1
      I_Contact( "Timer".T100.Q )
      wire#w2
      Coil( "A66" )
   END_RUNG
   RUNG wire#powerrail
      Contact( "Timer".T101.Q )
   END_RUNG wire#w1
   RUNG wire#powerrail
      Contact( "DB22_DisplayData".dbx22_2 )
   END_RUNG wire#w2
   // the same network as SCL:
   "A66" := (("In_Pos1" OR "Timer".T101.Q) AND NOT "Timer".T100.Q) OR "DB22_DisplayData".dbx22_2;
END_REGION

REGION Network 10: Conveyor pos1 motor
   RUNG wire#powerrail
      Contact( "V50_1" )
      Contact( "E121" )
      wire#w1
      Contact( "V15_6" )
      wire#w2
      Contact( "V90_7" )
      wire#w3
      Coil( "DB10_ExtConveyors".Out_ConvPos1 )
   END_RUNG
   RUNG wire#w1
      Contact( "DB22_DisplayData".dbx20_3 )
   END_RUNG wire#w2
   RUNG wire#powerrail
      Contact( "A34" )
      Contact( "E43" )
      Contact( "V90_7" )
   END_RUNG wire#w2
   RUNG wire#powerrail
      Contact( "DB22_DisplayData".dbx20_3 )
      I_Contact( "V50_1" )
      I_Contact( "E43" )
      I_Contact( "In_Pos1" )
   END_RUNG wire#w3
   // the same network as SCL:
   "DB10_ExtConveyors".Out_ConvPos1 := ((("V50_1" AND "E121" AND ("V15_6" OR "DB22_DisplayData".dbx20_3)) OR ("A34" AND "E43" AND "V90_7")) AND "V90_7") OR ("DB22_DisplayData".dbx20_3 AND NOT "V50_1" AND NOT "E43" AND NOT "In_Pos1");
END_REGION

REGION Network 11: Conveyor pos1 motor speed selection
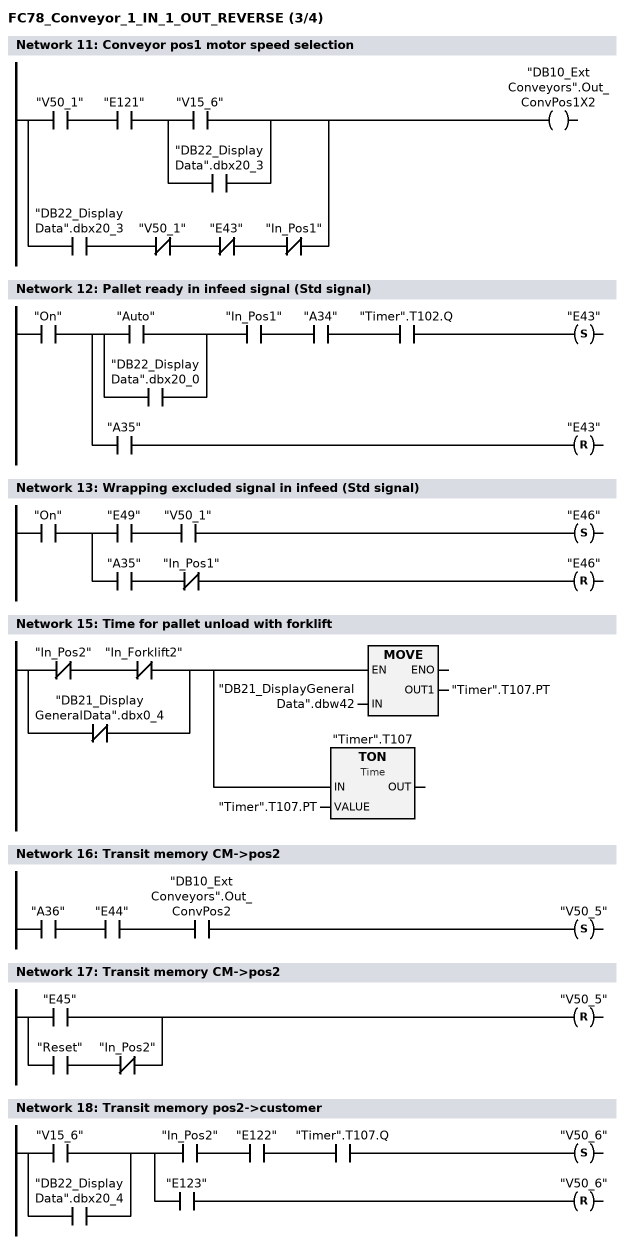
   RUNG wire#powerrail
      Contact( "V50_1" )
      Contact( "E121" )
      wire#w1
      Contact( "V15_6" )
      wire#w2
      Coil( "DB10_ExtConveyors".Out_ConvPos1X2 )
   END_RUNG
   RUNG wire#w1
      Contact( "DB22_DisplayData".dbx20_3 )
   END_RUNG wire#w2
   RUNG wire#powerrail
      Contact( "DB22_DisplayData".dbx20_3 )
      I_Contact( "V50_1" )
      I_Contact( "E43" )
      I_Contact( "In_Pos1" )
   END_RUNG wire#w2
   // the same network as SCL:
   "DB10_ExtConveyors".Out_ConvPos1X2 := ("V50_1" AND "E121" AND ("V15_6" OR "DB22_DisplayData".dbx20_3)) OR ("DB22_DisplayData".dbx20_3 AND NOT "V50_1" AND NOT "E43" AND NOT "In_Pos1");
END_REGION

REGION Network 12: Pallet ready in infeed signal (Std signal)
   RUNG wire#powerrail
      Contact( "On" )
      wire#w1
      Contact( "Auto" )
      wire#w2
      Contact( "In_Pos1" )
      Contact( "A34" )
      Contact( "Timer".T102.Q )
      S_Coil( "E43" )
   END_RUNG
   RUNG wire#w1
      Contact( "DB22_DisplayData".dbx20_0 )
   END_RUNG wire#w2
   RUNG wire#w1
      Contact( "A35" )
      R_Coil( "E43" )
   END_RUNG
   // the same network as SCL:
   IF "On" AND ("Auto" OR "DB22_DisplayData".dbx20_0) AND "In_Pos1" AND "A34" AND "Timer".T102.Q THEN
       "E43" := TRUE;
   END_IF;
   IF "On" AND "A35" THEN "E43" := FALSE; END_IF;
END_REGION

REGION Network 13: Wrapping excluded signal in infeed (Std signal)
   RUNG wire#powerrail
      Contact( "On" )
      wire#w1
      Contact( "E49" )
      Contact( "V50_1" )
      S_Coil( "E46" )
   END_RUNG
   RUNG wire#w1
      Contact( "A35" )
      I_Contact( "In_Pos1" )
      R_Coil( "E46" )
   END_RUNG
   // the same network as SCL:
   IF "On" AND "E49" AND "V50_1" THEN "E46" := TRUE; END_IF;
   IF "On" AND "A35" AND NOT "In_Pos1" THEN "E46" := FALSE; END_IF;
END_REGION

REGION Network 14: >>>>>>> OUTFEED CONVEYOR <<<<<<<<
END_REGION

REGION Network 15: Time for pallet unload with forklift
   #_w1 := (NOT "In_Pos2" AND NOT "In_Forklift2") OR NOT "DB21_DisplayGeneralData".dbx0_4;
   IF #_w1 THEN "Timer".T107.PT := "DB21_DisplayGeneralData".dbw42; END_IF;
   "Timer".T107.TON(IN := #_w1, PT := "Timer".T107.PT);   // TON coil
END_REGION

REGION Network 16: Transit memory CM->pos2
   RUNG wire#powerrail
      Contact( "A36" )
      Contact( "E44" )
      Contact( "DB10_ExtConveyors".Out_ConvPos2 )
      S_Coil( "V50_5" )
   END_RUNG
   // the same network as SCL:
   IF "A36" AND "E44" AND "DB10_ExtConveyors".Out_ConvPos2 THEN "V50_5" := TRUE; END_IF;
END_REGION

REGION Network 17: Transit memory CM->pos2
   RUNG wire#powerrail
      Contact( "E45" )
      wire#w1
      R_Coil( "V50_5" )
   END_RUNG
   RUNG wire#powerrail
      Contact( "Reset" )
      I_Contact( "In_Pos2" )
   END_RUNG wire#w1
   // the same network as SCL:
   IF "E45" OR ("Reset" AND NOT "In_Pos2") THEN "V50_5" := FALSE; END_IF;
END_REGION

REGION Network 18: Transit memory pos2->customer
   RUNG wire#powerrail
      Contact( "V15_6" )
      wire#w1
      Contact( "In_Pos2" )
      Contact( "E122" )
      Contact( "Timer".T107.Q )
      S_Coil( "V50_6" )
   END_RUNG
   RUNG wire#powerrail
      Contact( "DB22_DisplayData".dbx20_4 )
   END_RUNG wire#w1
   RUNG wire#w1
      Contact( "E123" )
      R_Coil( "V50_6" )
   END_RUNG
   // the same network as SCL:
   #_w1 := "V15_6" OR "DB22_DisplayData".dbx20_4;
   IF #_w1 AND "In_Pos2" AND "E122" AND "Timer".T107.Q THEN "V50_6" := TRUE; END_IF;
   IF #_w1 AND "E123" THEN "V50_6" := FALSE; END_IF;
END_REGION

REGION Network 19: Ready to receive pallet from outfeed signal (Signal for Technoplat)
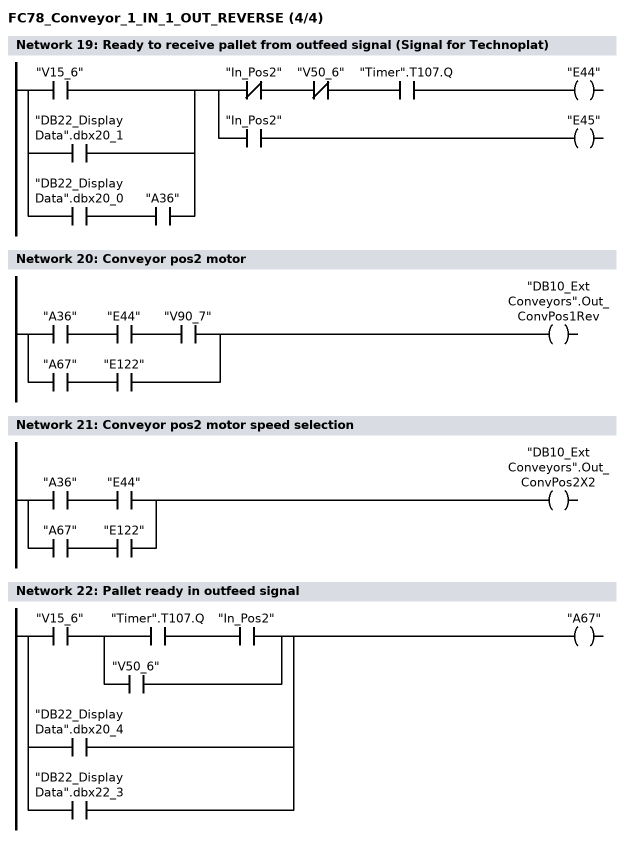
   RUNG wire#powerrail
      Contact( "V15_6" )
      wire#w1
      I_Contact( "In_Pos2" )
      I_Contact( "V50_6" )
      Contact( "Timer".T107.Q )
      Coil( "E44" )
   END_RUNG
   RUNG wire#powerrail
      Contact( "DB22_DisplayData".dbx20_1 )
   END_RUNG wire#w1
   RUNG wire#powerrail
      Contact( "DB22_DisplayData".dbx20_0 )
      Contact( "A36" )
   END_RUNG wire#w1
   RUNG wire#w1
      Contact( "In_Pos2" )
      Coil( "E45" )
   END_RUNG
   // the same network as SCL:
   #_w1 := "V15_6" OR "DB22_DisplayData".dbx20_1 OR ("DB22_DisplayData".dbx20_0 AND "A36");
   "E44" := #_w1 AND NOT "In_Pos2" AND NOT "V50_6" AND "Timer".T107.Q;
   "E45" := #_w1 AND "In_Pos2";
END_REGION

REGION Network 20: Conveyor pos2 motor
   RUNG wire#powerrail
      Contact( "A36" )
      Contact( "E44" )
      Contact( "V90_7" )
      wire#w1
      Coil( "DB10_ExtConveyors".Out_ConvPos1Rev )
   END_RUNG
   RUNG wire#powerrail
      Contact( "A67" )
      Contact( "E122" )
   END_RUNG wire#w1
   // the same network as SCL:
   "DB10_ExtConveyors".Out_ConvPos1Rev := ("A36" AND "E44" AND "V90_7") OR ("A67" AND "E122");
END_REGION

REGION Network 21: Conveyor pos2 motor speed selection
   RUNG wire#powerrail
      Contact( "A36" )
      Contact( "E44" )
      wire#w1
      Coil( "DB10_ExtConveyors".Out_ConvPos2X2 )
   END_RUNG
   RUNG wire#powerrail
      Contact( "A67" )
      Contact( "E122" )
   END_RUNG wire#w1
   // the same network as SCL:
   "DB10_ExtConveyors".Out_ConvPos2X2 := ("A36" AND "E44") OR ("A67" AND "E122");
END_REGION

REGION Network 22: Pallet ready in outfeed signal
   RUNG wire#powerrail
      Contact( "V15_6" )
      wire#w1
      Contact( "Timer".T107.Q )
      Contact( "In_Pos2" )
      wire#w2
      Coil( "A67" )
   END_RUNG
   RUNG wire#w1
      Contact( "V50_6" )
   END_RUNG wire#w2
   RUNG wire#powerrail
      Contact( "DB22_DisplayData".dbx20_4 )
   END_RUNG wire#w2
   RUNG wire#powerrail
      Contact( "DB22_DisplayData".dbx22_3 )
   END_RUNG wire#w2
   // the same network as SCL:
   "A67" := ("V15_6" AND (("Timer".T107.Q AND "In_Pos2") OR "V50_6")) OR "DB22_DisplayData".dbx20_4 OR "DB22_DisplayData".dbx22_3;
END_REGION
END_FUNCTION

FUNCTION "FC81_Optional" : Void   // FC81, LAD
TITLE = Optional
{ S7_Optimized_Access := 'TRUE' }
VERSION : 0.1
// stored: AutoNumber false, IsIECCheckEnabled false, SetENOAutomatically false, UDAEnableTagReadback false
BEGIN

REGION Network 1: Signal Automatic
